LIN {X 0,Y 545.057,Z 405.592,A -85,B 0,C 180,E1 -3721.915,E2 -3721.915} C_VEL
LIN {X 0,Y 545.061,Z 405.586,A -85,B 0,C 180,E1 -3724.565,E2 -3724.565} C_VEL
LIN {X 0,Y 545.033,Z 405.597,A -85,B 0,C 180,E1 -3727.304,E2 -3727.304} C_VEL
LIN {X 0,Y 545.067,Z 405.586,A -85,B 0,C 180,E1 -3730.143,E2 -3730.143} C_VEL
LIN {X 0,Y 545.05,Z 405.588,A -85,B 0,C 180,E1 -3732.695,E2 -3732.695} C_VEL
LIN {X 0,Y 545.063,Z 405.593,A -85,B 0,C 180,E1 -3735.167,E2 -3735.167} C_VEL
LIN {X 0,Y 545.08,Z 405.583,A -85,B 0,C 180,E1 -3737.897,E2 -3737.897} C_VEL
LIN {X 0,Y 545.083,Z 405.588,A -85,B 0,C 180,E1 -3740.818,E2 -3740.818} C_VEL
LIN {X 0,Y 545.045,Z 405.589,A -85,B 0,C 180,E1 -3743.62,E2 -3743.62} C_VEL
LIN {X 0,Y 545.069,Z 405.585,A -85,B 0,C 180,E1 -3746.328,E2 -3746.328} C_VEL
LIN {X 0,Y 545.069,Z 405.593,A -85,B 0,C 180,E1 -3748.952,E2 -3748.952} C_VEL
LIN {X 0,Y 545.087,Z 405.584,A -85,B 0,C 180,E1 -3751.507,E2 -3751.507} C_VEL
LIN {X 0,Y 545.089,Z 405.589,A -85,B 0,C 180,E1 -3754.493,E2 -3754.493} C_VEL
LIN {X 0,Y 545.041,Z 405.591,A -85,B 0,C 180,E1 -3757.242,E2 -3757.242} C_VEL
LIN {X 0,Y 545.119,Z 405.586,A -85,B 0,C 180,E1 -3760.415,E2 -3760.415} C_VEL
LIN {X 0,Y 545.048,Z 405.589,A -85,B 0,C 180,E1 -3763.52,E2 -3763.52} C_VEL
LIN {X 0,Y 545.109,Z 405.613,A -85,B 0,C 180,E1 -3765.555,E2 -3765.555} C_VEL
LIN {X 0,Y 546.501,Z 411.192,A -85,B 0,C 180,E1 -3765.668,E2 -3765.668} C_VEL
LIN {X 0,Y 546.206,Z 507.654,A -85,B 0,C 180,E1 -3766.963,E2 -3766.963} C_VEL
LIN {X 0,Y 546.091,Z 520.598,A -85,B 0,C 180,E1 -3767.268,E2 -3767.268} C_VEL
LIN {X 0,Y 545.891,Z 533.301,A -85,B 0,C 180,E1 -3767.735,E2 -3767.735} C_VEL
LIN {X 0,Y 545.749,Z 543.256,A -85,B 0,C 180,E1 -3768.218,E2 -3768.218} C_VEL
LIN {X 0,Y 545.618,Z 552.755,A -85,B 0,C 180,E1 -3768.79,E2 -3768.79} C_VEL
LIN {X 0,Y 545.433,Z 561.441,A -85,B 0,C 180,E1 -3769.42,E2 -3769.42} C_VEL
LIN {X 0,Y 545.222,Z 570.054,A -85,B 0,C 180,E1 -3770.166,E2 -3770.166} C_VEL
LIN {X 0,Y 545.101,Z 577.313,A -85,B 0,C 180,E1 -3770.913,E2 -3770.913} C_VEL
LIN {X 0,Y 544.944,Z 584.959,A -85,B 0,C 180,E1 -3771.844,E2 -3771.844} C_VEL
LIN {X 0,Y 544.822,Z 592.495,A -85,B 0,C 180,E1 -3772.961,E2 -3772.961} C_VEL
LIN {X 0,Y 544.778,Z 598.448,A -85,B 0,C 180,E1 -3774.076,E2 -3774.076} C_VEL
LIN {X 0,Y 544.628,Z 603.158,A -85,B 0,C 180,E1 -3775.189,E2 -3775.189} C_VEL
LIN {X 0,Y 544.669,Z 606.782,A -85,B 0,C 180,E1 -3776.301,E2 -3776.301} C_VEL
LIN {X 0,Y 544.65,Z 608.686,A -85,B 0,C 180,E1 -3777.041,E2 -3777.041} C_VEL
LIN {X 0,Y 544.571,Z 610.122,A -85,B 0,C 180,E1 -3777.781,E2 -3777.781} C_VEL
LIN {X 0,Y 544.542,Z 611.732,A -85,B 0,C 180,E1 -3779.261,E2 -3779.261} C_VEL
LIN {X 0,Y 544.542,Z 611.996,A -85,B 0,C 180,E1 -3780,E2 -3780} C_VEL
LIN {X 0,Y 544.546,Z 611.194,A -85,B 0,C 180,E1 -3781.479,E2 -3781.479} C_VEL
LIN {X 0,Y 544.572,Z 610.282,A -85,B 0,C 180,E1 -3782.219,E2 -3782.219} C_VEL
LIN {X 0,Y 544.651,Z 608.857,A -85,B 0,C 180,E1 -3782.959,E2 -3782.959} C_VEL
LIN {X 0,Y 544.66,Z 604.819,A -85,B 0,C 180,E1 -3784.44,E2 -3784.44} C_VEL
LIN {X 0,Y 544.737,Z 600.525,A -85,B 0,C 180,E1 -3785.553,E2 -3785.553} C_VEL
LIN {X 0,Y 544.753,Z 595.248,A -85,B 0,C 180,E1 -3786.632,E2 -3786.632} C_VEL
LIN {X 0,Y 544.85,Z 589.471,A -85,B 0,C 180,E1 -3787.598,E2 -3787.598} C_VEL
LIN {X 0,Y 544.991,Z 582.775,A -85,B 0,C 180,E1 -3788.528,E2 -3788.528} C_VEL
LIN {X 0,Y 545.142,Z 574.737,A -85,B 0,C 180,E1 -3789.461,E2 -3789.461} C_VEL
LIN {X 0,Y 545.384,Z 563.744,A -85,B 0,C 180,E1 -3790.487,E2 -3790.487} C_VEL
LIN {X 0,Y 545.553,Z 554.098,A -85,B 0,C 180,E1 -3791.211,E2 -3791.211} C_VEL
LIN {X 0,Y 545.718,Z 544.947,A -85,B 0,C 180,E1 -3791.778,E2 -3791.778} C_VEL
LIN {X 0,Y 545.842,Z 535.282,A -85,B 0,C 180,E1 -3792.266,E2 -3792.266} C_VEL
LIN {X 0,Y 545.982,Z 525.933,A -85,B 0,C 180,E1 -3792.64,E2 -3792.64} C_VEL
LIN {X 0,Y 546.169,Z 515.062,A -85,B 0,C 180,E1 -3792.967,E2 -3792.967} C_VEL
LIN {X 0,Y 546.272,Z 503.356,A -85,B 0,C 180,E1 -3793.201,E2 -3793.201} C_VEL
LIN {X 0,Y 546.42,Z 410.595,A -85,B 0,C 180,E1 -3794.432,E2 -3794.432} C_VEL
LIN {X 0,Y 545.081,Z 405.586,A -85,B 0,C 180,E1 -3794.538,E2 -3794.538} C_VEL
LIN {X 0,Y 545.063,Z 405.593,A -85,B 0,C 180,E1 -3797.417,E2 -3797.417} C_VEL
LIN {X 0,Y 545.094,Z 405.583,A -85,B 0,C 180,E1 -3800.372,E2 -3800.372} C_VEL
LIN {X 0,Y 545.058,Z 405.589,A -85,B 0,C 180,E1 -3803.353,E2 -3803.353} C_VEL
LIN {X 0,Y 544.433,Z 405.67,A -85,B 0,C 180,E1 -3803.97,E2 -3803.97} C_VEL
LIN {X 0,Y 541.586,Z 406.023,A -85,B 0,C 180,E1 -3804.971,E2 -3804.971} C_VEL
LIN {X 0,Y 539.155,Z 406.323,A -85,B 0,C 180,E1 -3805.777,E2 -3805.777} C_VEL
LIN {X 0,Y 538.11,Z 406.451,A -85,B 0,C 180,E1 -3806.4,E2 -3806.4} C_VEL
LIN {X 0,Y 538.026,Z 406.462,A -85,B 0,C 180,E1 -3806.611,E2 -3806.611} C_VEL
LIN {X 0,Y 538.033,Z 406.464,A -85,B 0,C 180,E1 -3808.933,E2 -3808.933} C_VEL
LIN {X 0,Y 538.013,Z 406.461,A -85,B 0,C 180,E1 -3811.887,E2 -3811.887} C_VEL
LIN {X 0,Y 538.015,Z 406.46,A -85,B 0,C 180,E1 -3814.618,E2 -3814.618} C_VEL
LIN {X 0,Y 538.008,Z 406.471,A -85,B 0,C 180,E1 -3817.17,E2 -3817.17} C_VEL
LIN {X 0,Y 538.026,Z 406.458,A -85,B 0,C 180,E1 -3819.797,E2 -3819.797} C_VEL
LIN {X 0,Y 538.023,Z 406.47,A -85,B 0,C 180,E1 -3822.786,E2 -3822.786} C_VEL
LIN {X 0,Y 538.027,Z 406.458,A -85,B 0,C 180,E1 -3825.926,E2 -3825.926} C_VEL
LIN {X 0,Y 538.051,Z 406.458,A -85,B 0,C 180,E1 -3829.224,E2 -3829.224} C_VEL
LIN {X 0,Y 537.991,Z 406.469,A -85,B 0,C 180,E1 -3832.122,E2 -3832.122} C_VEL
LIN {X 0,Y 537.997,Z 406.469,A -85,B 0,C 180,E1 -3834.915,E2 -3834.915} C_VEL
LIN {X 0,Y 538.021,Z 406.463,A -85,B 0,C 180,E1 -3837.617,E2 -3837.617} C_VEL
LIN {X 0,Y 538.003,Z 406.473,A -85,B 0,C 180,E1 -3840.238,E2 -3840.238} C_VEL
LIN {X 0,Y 538.004,Z 406.471,A -85,B 0,C 180,E1 -3842.793,E2 -3842.793} C_VEL
LIN {X 0,Y 538.05,Z 406.63,A -85,B 0,C 180,E1 -3845.845,E2 -3845.845} C_VEL
LIN {X 0,Y 539.322,Z 413.916,A -85,B 0,C 180,E1 -3846.987,E2 -3846.987} C_VEL
LIN {X 0,Y 539.029,Z 433.076,A -85,B 0,C 180,E1 -3849.844,E2 -3849.844} C_VEL
LIN {X 0,Y 538.696,Z 451.251,A -85,B 0,C 180,E1 -3852.538,E2 -3852.538} C_VEL
LIN {X 0,Y 538.403,Z 469.786,A -85,B 0,C 180,E1 -3855.289,E2 -3855.289} C_VEL
LIN {X 0,Y 539.611,Z 479.031,A -85,B 0,C 180,E1 -3855.452,E2 -3855.452} C_VEL
LIN {X 0,Y 539.309,Z 577.904,A -85,B 0,C 180,E1 -3856.794,E2 -3856.794} C_VEL
LIN {X 0,Y 539.12,Z 590.556,A -85,B 0,C 180,E1 -3857.1,E2 -3857.1} C_VEL
LIN {X 0,Y 538.931,Z 604.503,A -85,B 0,C 180,E1 -3857.622,E2 -3857.622} C_VEL
LIN {X 0,Y 538.715,Z 615.627,A -85,B 0,C 180,E1 -3858.196,E2 -3858.196} C_VEL
LIN {X 0,Y 538.565,Z 625.158,A -85,B 0,C 180,E1 -3858.807,E2 -3858.807} C_VEL
LIN {X 0,Y 538.391,Z 633.75,A -85,B 0,C 180,E1 -3859.47,E2 -3859.47} C_VEL
LIN {X 0,Y 538.137,Z 641.979,A -85,B 0,C 180,E1 -3860.225,E2 -3860.225} C_VEL
LIN {X 0,Y 538.032,Z 648.968,A -85,B 0,C 180,E1 -3860.982,E2 -3860.982} C_VEL
LIN {X 0,Y 537.861,Z 656.298,A -85,B 0,C 180,E1 -3861.925,E2 -3861.925} C_VEL
LIN {X 0,Y 537.744,Z 662.412,A -85,B 0,C 180,E1 -3862.868,E2 -3862.868} C_VEL
LIN {X 0,Y 537.651,Z 666.834,A -85,B 0,C 180,E1 -3863.667,E2 -3863.667} C_VEL
LIN {X 0,Y 537.587,Z 671.72,A -85,B 0,C 180,E1 -3864.749,E2 -3864.749} C_VEL
LIN {X 0,Y 537.603,Z 675.698,A -85,B 0,C 180,E1 -3865.877,E2 -3865.877} C_VEL
LIN {X 0,Y 537.551,Z 678.648,A -85,B 0,C 180,E1 -3867.002,E2 -3867.002} C_VEL
LIN {X 0,Y 537.49,Z 680.143,A -85,B 0,C 180,E1 -3867.752,E2 -3867.752} C_VEL
LIN {X 0,Y 537.442,Z 681.717,A -85,B 0,C 180,E1 -3869.251,E2 -3869.251} C_VEL
LIN {X 0,Y 537.442,Z 681.996,A -85,B 0,C 180,E1 -3870,E2 -3870} C_VEL
LIN {X 0,Y 537.452,Z 681.199,A -85,B 0,C 180,E1 -3871.499,E2 -3871.499} C_VEL
LIN {X 0,Y 537.49,Z 680.28,A -85,B 0,C 180,E1 -3872.248,E2 -3872.248} C_VEL
LIN {X 0,Y 537.591,Z 677.037,A -85,B 0,C 180,E1 -3873.748,E2 -3873.748} C_VEL
LIN {X 0,Y 537.54,Z 673.478,A -85,B 0,C 180,E1 -3874.875,E2 -3874.875} C_VEL
LIN {X 0,Y 537.672,Z 670.584,A -85,B 0,C 180,E1 -3875.626,E2 -3875.626} C_VEL
LIN {X 0,Y 537.706,Z 665.105,A -85,B 0,C 180,E1 -3876.756,E2 -3876.756} C_VEL
LIN {X 0,Y 537.829,Z 658.226,A -85,B 0,C 180,E1 -3877.886,E2 -3877.886} C_VEL
LIN {X 0,Y 537.956,Z 651.262,A -85,B 0,C 180,E1 -3878.83,E2 -3878.83} C_VEL
LIN {X 0,Y 538.11,Z 644.698,A -85,B 0,C 180,E1 -3879.586,E2 -3879.586} C_VEL
LIN {X 0,Y 538.274,Z 636.977,A -85,B 0,C 180,E1 -3880.342,E2 -3880.342} C_VEL
LIN {X 0,Y 538.501,Z 627.706,A -85,B 0,C 180,E1 -3881.099,E2 -3881.099} C_VEL
LIN {X 0,Y 538.688,Z 618.38,A -85,B 0,C 180,E1 -3881.729,E2 -3881.729} C_VEL
LIN {X 0,Y 538.849,Z 609.277,A -85,B 0,C 180,E1 -3882.236,E2 -3882.236} C_VEL
LIN {X 0,Y 539.03,Z 598.562,A -85,B 0,C 180,E1 -3882.71,E2 -3882.71} C_VEL
LIN {X 0,Y 539.178,Z 586.982,A -85,B 0,C 180,E1 -3883.09,E2 -3883.09} C_VEL
LIN {X 0,Y 539.35,Z 574.949,A -85,B 0,C 180,E1 -3883.349,E2 -3883.349} C_VEL
LIN {X 0,Y 539.633,Z 477.878,A -85,B 0,C 180,E1 -3884.653,E2 -3884.653} C_VEL
LIN {X 0,Y 538.415,Z 469.73,A -85,B 0,C 180,E1 -3884.811,E2 -3884.811} C_VEL
LIN {X 0,Y 538.775,Z 447.637,A -85,B 0,C 180,E1 -3888.09,E2 -3888.09} C_VEL
LIN {X 0,Y 539.079,Z 429.341,A -85,B 0,C 180,E1 -3890.809,E2 -3890.809} C_VEL
LIN {X 0,Y 539.333,Z 414.54,A -85,B 0,C 180,E1 -3893.012,E2 -3893.012} C_VEL
LIN {X 0,Y 538.002,Z 406.471,A -85,B 0,C 180,E1 -3894.298,E2 -3894.298} C_VEL
LIN {X 0,Y 538.003,Z 406.471,A -85,B 0,C 180,E1 -3897.34,E2 -3897.34} C_VEL
LIN {X 0,Y 538.003,Z 406.473,A -85,B 0,C 180,E1 -3899.762,E2 -3899.762} C_VEL
LIN {X 0,Y 538.021,Z 406.464,A -85,B 0,C 180,E1 -3902.383,E2 -3902.383} C_VEL
LIN {X 0,Y 537.997,Z 406.471,A -85,B 0,C 180,E1 -3905.085,E2 -3905.085} C_VEL
LIN {X 0,Y 537.992,Z 406.468,A -85,B 0,C 180,E1 -3907.878,E2 -3907.878} C_VEL
LIN {X 0,Y 538.051,Z 406.46,A -85,B 0,C 180,E1 -3910.776,E2 -3910.776} C_VEL
LIN {X 0,Y 538.034,Z 406.459,A -85,B 0,C 180,E1 -3914.075,E2 -3914.075} C_VEL
LIN {X 0,Y 538.029,Z 406.468,A -85,B 0,C 180,E1 -3917.012,E2 -3917.012} C_VEL
LIN {X 0,Y 538.052,Z 406.462,A -85,B 0,C 180,E1 -3919.253,E2 -3919.253} C_VEL
LIN {X 0,Y 537.993,Z 406.467,A -85,B 0,C 180,E1 -3922.122,E2 -3922.122} C_VEL
LIN {X 0,Y 537.998,Z 406.47,A -85,B 0,C 180,E1 -3924.915,E2 -3924.915} C_VEL
LIN {X 0,Y 538.021,Z 406.462,A -85,B 0,C 180,E1 -3927.617,E2 -3927.617} C_VEL
LIN {X 0,Y 538.003,Z 406.47,A -85,B 0,C 180,E1 -3930.238,E2 -3930.238} C_VEL
LIN {X 0,Y 538.013,Z 406.468,A -85,B 0,C 180,E1 -3932.793,E2 -3932.793} C_VEL
LIN {X 0,Y 538.018,Z 406.563,A -85,B 0,C 180,E1 -3935.815,E2 -3935.815} C_VEL
LIN {X 0,Y 539.339,Z 414.074,A -85,B 0,C 180,E1 -3936.988,E2 -3936.988} C_VEL
LIN {X 0,Y 539.05,Z 431.921,A -85,B 0,C 180,E1 -3939.679,E2 -3939.679} C_VEL
LIN {X 0,Y 538.681,Z 452.563,A -85,B 0,C 180,E1 -3942.734,E2 -3942.734} C_VEL
LIN {X 0,Y 538.404,Z 469.886,A -85,B 0,C 180,E1 -3945.304,E2 -3945.304} C_VEL
LIN {X 0,Y 539.606,Z 478.79,A -85,B 0,C 180,E1 -3945.455,E2 -3945.455} C_VEL
LIN {X 0,Y 539.3,Z 576.13,A -85,B 0,C 180,E1 -3946.769,E2 -3946.769} C_VEL
LIN {X 0,Y 539.191,Z 586.049,A -85,B 0,C 180,E1 -3946.982,E2 -3946.982} C_VEL
LIN {X 0,Y 539.057,Z 596.036,A -85,B 0,C 180,E1 -3947.29,E2 -3947.29} C_VEL
LIN {X 0,Y 538.879,Z 605.384,A -85,B 0,C 180,E1 -3947.669,E2 -3947.669} C_VEL
LIN {X 0,Y 538.733,Z 615.228,A -85,B 0,C 180,E1 -3948.174,E2 -3948.174} C_VEL
LIN {X 0,Y 538.592,Z 623.796,A -85,B 0,C 180,E1 -3948.712,E2 -3948.712} C_VEL
LIN {X 0,Y 538.369,Z 632.608,A -85,B 0,C 180,E1 -3949.374,E2 -3949.374} C_VEL
LIN {X 0,Y 538.213,Z 640.052,A -85,B 0,C 180,E1 -3950.037,E2 -3950.037} C_VEL
LIN {X 0,Y 538.056,Z 647.305,A -85,B 0,C 180,E1 -3950.793,E2 -3950.793} C_VEL
LIN {X 0,Y 537.884,Z 654.929,A -85,B 0,C 180,E1 -3951.736,E2 -3951.736} C_VEL
LIN {X 0,Y 537.759,Z 661.273,A -85,B 0,C 180,E1 -3952.679,E2 -3952.679} C_VEL
LIN {X 0,Y 537.639,Z 666.854,A -85,B 0,C 180,E1 -3953.679,E2 -3953.679} C_VEL
LIN {X 0,Y 537.586,Z 671.701,A -85,B 0,C 180,E1 -3954.749,E2 -3954.749} C_VEL
LIN {X 0,Y 537.604,Z 675.701,A -85,B 0,C 180,E1 -3955.877,E2 -3955.877} C_VEL
LIN {X 0,Y 537.551,Z 678.665,A -85,B 0,C 180,E1 -3957.002,E2 -3957.002} C_VEL
LIN {X 0,Y 537.451,Z 681.145,A -85,B 0,C 180,E1 -3958.501,E2 -3958.501} C_VEL
LIN {X 0,Y 537.442,Z 681.741,A -85,B 0,C 180,E1 -3959.251,E2 -3959.251} C_VEL
LIN {X 0,Y 537.442,Z 681.806,A -85,B 0,C 180,E1 -3960.749,E2 -3960.749} C_VEL
LIN {X 0,Y 537.452,Z 681.221,A -85,B 0,C 180,E1 -3961.499,E2 -3961.499} C_VEL
LIN {X 0,Y 537.552,Z 678.878,A -85,B 0,C 180,E1 -3962.998,E2 -3962.998} C_VEL
LIN {X 0,Y 537.604,Z 675.992,A -85,B 0,C 180,E1 -3964.123,E2 -3964.123} C_VEL
LIN {X 0,Y 537.587,Z 672.073,A -85,B 0,C 180,E1 -3965.251,E2 -3965.251} C_VEL
LIN {X 0,Y 537.639,Z 667.317,A -85,B 0,C 180,E1 -3966.32,E2 -3966.32} C_VEL
LIN {X 0,Y 537.754,Z 661.829,A -85,B 0,C 180,E1 -3967.321,E2 -3967.321} C_VEL
LIN {X 0,Y 537.875,Z 655.592,A -85,B 0,C 180,E1 -3968.264,E2 -3968.264} C_VEL
LIN {X 0,Y 537.982,Z 649.743,A -85,B 0,C 180,E1 -3969.019,E2 -3969.019} C_VEL
LIN {X 0,Y 538.129,Z 642.926,A -85,B 0,C 180,E1 -3969.775,E2 -3969.775} C_VEL
LIN {X 0,Y 538.373,Z 633.697,A -85,B 0,C 180,E1 -3970.626,E2 -3970.626} C_VEL
LIN {X 0,Y 538.555,Z 625.09,A -85,B 0,C 180,E1 -3971.288,E2 -3971.288} C_VEL
LIN {X 0,Y 538.741,Z 616.029,A -85,B 0,C 180,E1 -3971.869,E2 -3971.869} C_VEL
LIN {X 0,Y 538.893,Z 606.287,A -85,B 0,C 180,E1 -3972.379,E2 -3972.379} C_VEL
LIN {X 0,Y 539.029,Z 597.178,A -85,B 0,C 180,E1 -3972.758,E2 -3972.758} C_VEL
LIN {X 0,Y 539.161,Z 587.581,A -85,B 0,C 180,E1 -3973.066,E2 -3973.066} C_VEL
LIN {X 0,Y 539.294,Z 577.096,A -85,B 0,C 180,E1 -3973.303,E2 -3973.303} C_VEL
LIN {X 0,Y 539.655,Z 478.373,A -85,B 0,C 180,E1 -3974.639,E2 -3974.639} C_VEL
LIN {X 0,Y 538.411,Z 469.814,A -85,B 0,C 180,E1 -3974.798,E2 -3974.798} C_VEL
LIN {X 0,Y 538.633,Z 454.436,A -85,B 0,C 180,E1 -3977.072,E2 -3977.072} C_VEL
LIN {X 0,Y 539.039,Z 434.478,A -85,B 0,C 180,E1 -3980.04,E2 -3980.04} C_VEL
LIN {X 0,Y 539.172,Z 413.599,A -85,B 0,C 180,E1 -3983.02,E2 -3983.02} C_VEL
LIN {X 0,Y 538.022,Z 406.471,A -85,B 0,C 180,E1 -3984.1,E2 -3984.1} C_VEL
LIN {X 0,Y 538.003,Z 406.47,A -85,B 0,C 180,E1 -3987.207,E2 -3987.207} C_VEL
LIN {X 0,Y 538.003,Z 406.473,A -85,B 0,C 180,E1 -3989.762,E2 -3989.762} C_VEL
LIN {X 0,Y 538.021,Z 406.464,A -85,B 0,C 180,E1 -3992.383,E2 -3992.383} C_VEL
LIN {X 0,Y 537.997,Z 406.471,A -85,B 0,C 180,E1 -3995.085,E2 -3995.085} C_VEL
LIN {X 0,Y 537.992,Z 406.468,A -85,B 0,C 180,E1 -3997.878,E2 -3997.878} C_VEL
LIN {X 0,Y 538.051,Z 406.463,A -85,B 0,C 180,E1 -4000.776,E2 -4000.776} C_VEL
LIN {X 0,Y 538.033,Z 406.462,A -85,B 0,C 180,E1 -4004.075,E2 -4004.075} C_VEL
LIN {X 0,Y 538.029,Z 406.468,A -85,B 0,C 180,E1 -4007.012,E2 -4007.012} C_VEL
LIN {X 0,Y 538.051,Z 406.462,A -85,B 0,C 180,E1 -4009.253,E2 -4009.253} C_VEL
LIN {X 0,Y 537.992,Z 406.468,A -85,B 0,C 180,E1 -4012.122,E2 -4012.122} C_VEL
LIN {X 0,Y 537.997,Z 406.471,A -85,B 0,C 180,E1 -4014.915,E2 -4014.915} C_VEL
LIN {X 0,Y 538.021,Z 406.463,A -85,B 0,C 180,E1 -4017.617,E2 -4017.617} C_VEL
LIN {X 0,Y 538.002,Z 406.472,A -85,B 0,C 180,E1 -4020.238,E2 -4020.238} C_VEL
LIN {X 0,Y 538.07,Z 406.661,A -85,B 0,C 180,E1 -4023.347,E2 -4023.347} C_VEL
LIN {X 0,Y 539.845,Z 415.143,A -85,B 0,C 180,E1 -4024.557,E2 -4024.557} C_VEL
LIN {X 0,Y 539.721,Z 432.182,A -85,B 0,C 180,E1 -4026.802,E2 -4026.802} C_VEL
LIN {X 0,Y 539.23,Z 454.329,A -85,B 0,C 180,E1 -4029.653,E2 -4029.653} C_VEL
LIN {X 0,Y 538.822,Z 478.604,A -85,B 0,C 180,E1 -4032.738,E2 -4032.738} C_VEL
LIN {X 0,Y 538.509,Z 498.569,A -85,B 0,C 180,E1 -4035.244,E2 -4035.244} C_VEL
LIN {X 0,Y 539.647,Z 507.696,A -85,B 0,C 180,E1 -4035.395,E2 -4035.395} C_VEL
LIN {X 0,Y 539.307,Z 607.943,A -85,B 0,C 180,E1 -4036.746,E2 -4036.746} C_VEL
LIN {X 0,Y 539.114,Z 621.214,A -85,B 0,C 180,E1 -4037.076,E2 -4037.076} C_VEL
LIN {X 0,Y 538.933,Z 633.367,A -85,B 0,C 180,E1 -4037.527,E2 -4037.527} C_VEL
LIN {X 0,Y 538.742,Z 645.405,A -85,B 0,C 180,E1 -4038.13,E2 -4038.13} C_VEL
LIN {X 0,Y 538.506,Z 657.192,A -85,B 0,C 180,E1 -4038.901,E2 -4038.901} C_VEL
LIN {X 0,Y 538.261,Z 667.604,A -85,B 0,C 180,E1 -4039.753,E2 -4039.753} C_VEL
LIN {X 0,Y 538.068,Z 676.113,A -85,B 0,C 180,E1 -4040.603,E2 -4040.603} C_VEL
LIN {X 0,Y 537.921,Z 683.96,A -85,B 0,C 180,E1 -4041.548,E2 -4041.548} C_VEL
LIN {X 0,Y 537.755,Z 691.621,A -85,B 0,C 180,E1 -4042.679,E2 -4042.679} C_VEL
LIN {X 0,Y 537.693,Z 698.679,A -85,B 0,C 180,E1 -4043.998,E2 -4043.998} C_VEL
LIN {X 0,Y 537.54,Z 703.373,A -85,B 0,C 180,E1 -4045.125,E2 -4045.125} C_VEL
LIN {X 0,Y 537.591,Z 706.958,A -85,B 0,C 180,E1 -4046.252,E2 -4046.252} C_VEL
LIN {X 0,Y 537.551,Z 708.807,A -85,B 0,C 180,E1 -4047.002,E2 -4047.002} C_VEL
LIN {X 0,Y 537.451,Z 711.182,A -85,B 0,C 180,E1 -4048.501,E2 -4048.501} C_VEL
LIN {X 0,Y 537.442,Z 712,A -85,B 0,C 180,E1 -4050,E2 -4050} C_VEL
LIN {X 0,Y 537.451,Z 711.184,A -85,B 0,C 180,E1 -4051.499,E2 -4051.499} C_VEL
LIN {X 0,Y 537.551,Z 708.81,A -85,B 0,C 180,E1 -4052.998,E2 -4052.998} C_VEL
LIN {X 0,Y 537.603,Z 705.895,A -85,B 0,C 180,E1 -4054.123,E2 -4054.123} C_VEL
LIN {X 0,Y 537.587,Z 701.948,A -85,B 0,C 180,E1 -4055.251,E2 -4055.251} C_VEL
LIN {X 0,Y 537.651,Z 697.08,A -85,B 0,C 180,E1 -4056.335,E2 -4056.335} C_VEL
LIN {X 0,Y 537.791,Z 690.466,A -85,B 0,C 180,E1 -4057.509,E2 -4057.509} C_VEL
LIN {X 0,Y 537.972,Z 682.477,A -85,B 0,C 180,E1 -4058.641,E2 -4058.641} C_VEL
LIN {X 0,Y 538.145,Z 674.332,A -85,B 0,C 180,E1 -4059.585,E2 -4059.585} C_VEL
LIN {X 0,Y 538.366,Z 664.396,A -85,B 0,C 180,E1 -4060.531,E2 -4060.531} C_VEL
LIN {X 0,Y 538.583,Z 654.591,A -85,B 0,C 180,E1 -4061.288,E2 -4061.288} C_VEL
LIN {X 0,Y 538.745,Z 643.853,A -85,B 0,C 180,E1 -4061.956,E2 -4061.956} C_VEL
LIN {X 0,Y 538.979,Z 631.099,A -85,B 0,C 180,E1 -4062.568,E2 -4062.568} C_VEL
LIN {X 0,Y 539.17,Z 618.083,A -85,B 0,C 180,E1 -4063.018,E2 -4063.018} C_VEL
LIN {X 0,Y 539.32,Z 605.098,A -85,B 0,C 180,E1 -4063.302,E2 -4063.302} C_VEL
LIN {X 0,Y 539.592,Z 506.19,A -85,B 0,C 180,E1 -4064.624,E2 -4064.624} C_VEL
LIN {X 0,Y 538.478,Z 498.265,A -85,B 0,C 180,E1 -4064.774,E2 -4064.774} C_VEL
LIN {X 0,Y 538.849,Z 473.854,A -85,B 0,C 180,E1 -4067.803,E2 -4067.803} C_VEL
LIN {X 0,Y 539.201,Z 451.45,A -85,B 0,C 180,E1 -4070.605,E2 -4070.605} C_VEL
LIN {X 0,Y 539.464,Z 427.686,A -85,B 0,C 180,E1 -4073.616,E2 -4073.616} C_VEL
LIN {X 0,Y 539.64,Z 414.953,A -85,B 0,C 180,E1 -4075.247,E2 -4075.247} C_VEL
LIN {X 0,Y 538.006,Z 406.469,A -85,B 0,C 180,E1 -4076.421,E2 -4076.421} C_VEL
LIN {X 0,Y 537.994,Z 406.469,A -85,B 0,C 180,E1 -4078.926,E2 -4078.926} C_VEL
LIN {X 0,Y 538.012,Z 406.47,A -85,B 0,C 180,E1 -4081.887,E2 -4081.887} C_VEL
LIN {X 0,Y 538.01,Z 406.465,A -85,B 0,C 180,E1 -4084.617,E2 -4084.617} C_VEL
LIN {X 0,Y 538.001,Z 406.471,A -85,B 0,C 180,E1 -4087.169,E2 -4087.169} C_VEL
LIN {X 0,Y 538.024,Z 406.466,A -85,B 0,C 180,E1 -4089.797,E2 -4089.797} C_VEL
LIN {X 0,Y 538.002,Z 406.467,A -85,B 0,C 180,E1 -4092.788,E2 -4092.788} C_VEL
LIN {X 0,Y 538.028,Z 406.469,A -85,B 0,C 180,E1 -4095.14,E2 -4095.14} C_VEL
LIN {X 0,Y 538.033,Z 406.461,A -85,B 0,C 180,E1 -4098.227,E2 -4098.227} C_VEL
LIN {X 0,Y 538.016,Z 406.47,A -85,B 0,C 180,E1 -4101.17,E2 -4101.17} C_VEL
LIN {X 0,Y 537.997,Z 406.465,A -85,B 0,C 180,E1 -4104.089,E2 -4104.089} C_VEL
LIN {X 0,Y 538.033,Z 406.466,A -85,B 0,C 180,E1 -4106.727,E2 -4106.727} C_VEL
LIN {X 0,Y 538.03,Z 406.463,A -85,B 0,C 180,E1 -4109.556,E2 -4109.556} C_VEL
LIN {X 0,Y 538.053,Z 406.467,A -85,B 0,C 180,E1 -4112.65,E2 -4112.65} C_VEL
LIN {X 0,Y 538.027,Z 406.466,A -85,B 0,C 180,E1 -4115.291,E2 -4115.291} C_VEL
LIN {X 0,Y 538.019,Z 406.466,A -85,B 0,C 180,E1 -4118.042,E2 -4118.042} C_VEL
LIN {X 0,Y 538.083,Z 406.459,A -85,B 0,C 180,E1 -4120.148,E2 -4120.148} C_VEL
LIN {X 0,Y 537.999,Z 406.468,A -85,B 0,C 180,E1 -4123.298,E2 -4123.298} C_VEL
LIN {X 0,Y 538.088,Z 406.459,A -85,B 0,C 180,E1 -4125.362,E2 -4125.362} C_VEL
LIN {X 0,Y 539.715,Z 412.557,A -85,B 0,C 180,E1 -4125.498,E2 -4125.498} C_VEL
LIN {X 0,Y 539.295,Z 508.582,A -85,B 0,C 180,E1 -4126.817,E2 -4126.817} C_VEL
LIN {X 0,Y 539.156,Z 521.366,A -85,B 0,C 180,E1 -4127.125,E2 -4127.125} C_VEL
LIN {X 0,Y 538.935,Z 534.56,A -85,B 0,C 180,E1 -4127.622,E2 -4127.622} C_VEL
LIN {X 0,Y 538.801,Z 543.956,A -85,B 0,C 180,E1 -4128.089,E2 -4128.089} C_VEL
LIN {X 0,Y 538.639,Z 554.039,A -85,B 0,C 180,E1 -4128.713,E2 -4128.713} C_VEL
LIN {X 0,Y 538.45,Z 562.824,A -85,B 0,C 180,E1 -4129.376,E2 -4129.376} C_VEL
LIN {X 0,Y 538.213,Z 570.225,A -85,B 0,C 180,E1 -4130.037,E2 -4130.037} C_VEL
LIN {X 0,Y 538.081,Z 577.418,A -85,B 0,C 180,E1 -4130.793,E2 -4130.793} C_VEL
LIN {X 0,Y 537.918,Z 583.561,A -85,B 0,C 180,E1 -4131.548,E2 -4131.548} C_VEL
LIN {X 0,Y 537.756,Z 591.312,A -85,B 0,C 180,E1 -4132.679,E2 -4132.679} C_VEL
LIN {X 0,Y 537.694,Z 598.443,A -85,B 0,C 180,E1 -4133.998,E2 -4133.998} C_VEL
LIN {X 0,Y 537.54,Z 603.153,A -85,B 0,C 180,E1 -4135.125,E2 -4135.125} C_VEL
LIN {X 0,Y 537.591,Z 606.777,A -85,B 0,C 180,E1 -4136.252,E2 -4136.252} C_VEL
LIN {X 0,Y 537.551,Z 608.682,A -85,B 0,C 180,E1 -4137.002,E2 -4137.002} C_VEL
LIN {X 0,Y 537.49,Z 610.118,A -85,B 0,C 180,E1 -4137.752,E2 -4137.752} C_VEL
LIN {X 0,Y 537.442,Z 611.725,A -85,B 0,C 180,E1 -4139.251,E2 -4139.251} C_VEL
LIN {X 0,Y 537.442,Z 611.996,A -85,B 0,C 180,E1 -4140,E2 -4140} C_VEL
LIN {X 0,Y 537.452,Z 611.187,A -85,B 0,C 180,E1 -4141.499,E2 -4141.499} C_VEL
LIN {X 0,Y 537.49,Z 610.28,A -85,B 0,C 180,E1 -4142.248,E2 -4142.248} C_VEL
LIN {X 0,Y 537.552,Z 608.85,A -85,B 0,C 180,E1 -4142.998,E2 -4142.998} C_VEL
LIN {X 0,Y 537.557,Z 604.809,A -85,B 0,C 180,E1 -4144.499,E2 -4144.499} C_VEL
LIN {X 0,Y 537.671,Z 600.515,A -85,B 0,C 180,E1 -4145.626,E2 -4145.626} C_VEL
LIN {X 0,Y 537.682,Z 595.743,A -85,B 0,C 180,E1 -4146.627,E2 -4146.627} C_VEL
LIN {X 0,Y 537.799,Z 589.459,A -85,B 0,C 180,E1 -4147.698,E2 -4147.698} C_VEL
LIN {X 0,Y 537.951,Z 582.797,A -85,B 0,C 180,E1 -4148.641,E2 -4148.641} C_VEL
LIN {X 0,Y 538.131,Z 574.833,A -85,B 0,C 180,E1 -4149.585,E2 -4149.585} C_VEL
LIN {X 0,Y 538.387,Z 563.89,A -85,B 0,C 180,E1 -4150.625,E2 -4150.625} C_VEL
LIN {X 0,Y 538.563,Z 555.302,A -85,B 0,C 180,E1 -4151.288,E2 -4151.288} C_VEL
LIN {X 0,Y 538.764,Z 544.938,A -85,B 0,C 180,E1 -4151.943,E2 -4151.943} C_VEL
LIN {X 0,Y 538.911,Z 534.391,A -85,B 0,C 180,E1 -4152.474,E2 -4152.474} C_VEL
LIN {X 0,Y 539.183,Z 521.951,A -85,B 0,C 180,E1 -4152.946,E2 -4152.946} C_VEL
LIN {X 0,Y 539.274,Z 509.732,A -85,B 0,C 180,E1 -4153.255,E2 -4153.255} C_VEL
LIN {X 0,Y 539.454,Z 479.835,A -85,B 0,C 180,E1 -4153.682,E2 -4153.682} C_VEL
LIN {X 0,Y 539.592,Z 411.558,A -85,B 0,C 180,E1 -4154.605,E2 -4154.605} C_VEL
LIN {X 0,Y 538.059,Z 406.461,A -85,B 0,C 180,E1 -4154.736,E2 -4154.736} C_VEL
LIN {X 0,Y 538.015,Z 406.472,A -85,B 0,C 180,E1 -4157.524,E2 -4157.524} C_VEL
LIN {X 0,Y 538.088,Z 406.459,A -85,B 0,C 180,E1 -4159.881,E2 -4159.881} C_VEL
LIN {X 0,Y 538.014,Z 406.467,A -85,B 0,C 180,E1 -4163.072,E2 -4163.072} C_VEL
LIN {X 0,Y 538.033,Z 406.46,A -85,B 0,C 180,E1 -4166.367,E2 -4166.367} C_VEL
LIN {X 0,Y 538.026,Z 406.462,A -85,B 0,C 180,E1 -4166.611,E2 -4166.611} C_VEL
LIN {X 0,Y 537.359,Z 406.552,A -85,B 0,C 180,E1 -4167.235,E2 -4167.235} C_VEL
LIN {X 0,Y 534.492,Z 406.908,A -85,B 0,C 180,E1 -4168.249,E2 -4168.249} C_VEL
LIN {X 0,Y 532.073,Z 407.208,A -85,B 0,C 180,E1 -4169.066,E2 -4169.066} C_VEL
LIN {X 0,Y 531.042,Z 407.335,A -85,B 0,C 180,E1 -4169.696,E2 -4169.696} C_VEL
LIN {X 0,Y 530.962,Z 407.342,A -85,B 0,C 180,E1 -4169.91,E2 -4169.91} C_VEL
LIN {X 0,Y 530.97,Z 407.343,A -85,B 0,C 180,E1 -4172.867,E2 -4172.867} C_VEL
LIN {X 0,Y 530.957,Z 407.344,A -85,B 0,C 180,E1 -4175.62,E2 -4175.62} C_VEL
LIN {X 0,Y 530.97,Z 407.345,A -85,B 0,C 180,E1 -4178.654,E2 -4178.654} C_VEL
LIN {X 0,Y 530.997,Z 407.339,A -85,B 0,C 180,E1 -4181.436,E2 -4181.436} C_VEL
LIN {X 0,Y 530.989,Z 407.344,A -85,B 0,C 180,E1 -4184.547,E2 -4184.547} C_VEL
LIN {X 0,Y 530.985,Z 407.339,A -85,B 0,C 180,E1 -4187.834,E2 -4187.834} C_VEL
LIN {X 0,Y 530.988,Z 407.343,A -85,B 0,C 180,E1 -4190.556,E2 -4190.556} C_VEL
LIN {X 0,Y 530.953,Z 407.342,A -85,B 0,C 180,E1 -4193.441,E2 -4193.441} C_VEL
LIN {X 0,Y 531.002,Z 407.344,A -85,B 0,C 180,E1 -4196.494,E2 -4196.494} C_VEL
LIN {X 0,Y 530.964,Z 407.343,A -85,B 0,C 180,E1 -4199.357,E2 -4199.357} C_VEL
LIN {X 0,Y 530.963,Z 407.351,A -85,B 0,C 180,E1 -4202.479,E2 -4202.479} C_VEL
LIN {X 0,Y 531.015,Z 407.464,A -85,B 0,C 180,E1 -4205.673,E2 -4205.673} C_VEL
LIN {X 0,Y 532.36,Z 415.042,A -85,B 0,C 180,E1 -4206.874,E2 -4206.874} C_VEL
LIN {X 0,Y 532.068,Z 433.71,A -85,B 0,C 180,E1 -4209.69,E2 -4209.69} C_VEL
LIN {X 0,Y 531.696,Z 453.83,A -85,B 0,C 180,E1 -4212.698,E2 -4212.698} C_VEL
LIN {X 0,Y 531.409,Z 469.902,A -85,B 0,C 180,E1 -4215.092,E2 -4215.092} C_VEL
LIN {X 0,Y 532.745,Z 479.269,A -85,B 0,C 180,E1 -4215.262,E2 -4215.262} C_VEL
LIN {X 0,Y 532.414,Z 578.141,A -85,B 0,C 180,E1 -4216.619,E2 -4216.619} C_VEL
LIN {X 0,Y 532.207,Z 591.571,A -85,B 0,C 180,E1 -4216.954,E2 -4216.954} C_VEL
LIN {X 0,Y 532,Z 604.658,A -85,B 0,C 180,E1 -4217.458,E2 -4217.458} C_VEL
LIN {X 0,Y 531.79,Z 616.926,A -85,B 0,C 180,E1 -4218.099,E2 -4218.099} C_VEL
LIN {X 0,Y 531.549,Z 628.024,A -85,B 0,C 180,E1 -4218.851,E2 -4218.851} C_VEL
LIN {X 0,Y 531.227,Z 639.261,A -85,B 0,C 180,E1 -4219.808,E2 -4219.808} C_VEL
LIN {X 0,Y 531.023,Z 647.488,A -85,B 0,C 180,E1 -4220.67,E2 -4220.67} C_VEL
LIN {X 0,Y 530.851,Z 655.076,A -85,B 0,C 180,E1 -4221.626,E2 -4221.626} C_VEL
LIN {X 0,Y 530.672,Z 662.446,A -85,B 0,C 180,E1 -4222.772,E2 -4222.772} C_VEL
LIN {X 0,Y 530.564,Z 667.294,A -85,B 0,C 180,E1 -4223.681,E2 -4223.681} C_VEL
LIN {X 0,Y 530.524,Z 671.716,A -85,B 0,C 180,E1 -4224.679,E2 -4224.679} C_VEL
LIN {X 0,Y 530.523,Z 675.693,A -85,B 0,C 180,E1 -4225.822,E2 -4225.822} C_VEL
LIN {X 0,Y 530.457,Z 678.641,A -85,B 0,C 180,E1 -4226.962,E2 -4226.962} C_VEL
LIN {X 0,Y 530.411,Z 680.144,A -85,B 0,C 180,E1 -4227.722,E2 -4227.722} C_VEL
LIN {X 0,Y 530.344,Z 681.709,A -85,B 0,C 180,E1 -4229.241,E2 -4229.241} C_VEL
LIN {X 0,Y 530.343,Z 681.997,A -85,B 0,C 180,E1 -4230,E2 -4230} C_VEL
LIN {X 0,Y 530.361,Z 681.191,A -85,B 0,C 180,E1 -4231.519,E2 -4231.519} C_VEL
LIN {X 0,Y 530.411,Z 680.281,A -85,B 0,C 180,E1 -4232.278,E2 -4232.278} C_VEL
LIN {X 0,Y 530.516,Z 677.029,A -85,B 0,C 180,E1 -4233.798,E2 -4233.798} C_VEL
LIN {X 0,Y 530.458,Z 673.469,A -85,B 0,C 180,E1 -4234.94,E2 -4234.94} C_VEL
LIN {X 0,Y 530.605,Z 670.581,A -85,B 0,C 180,E1 -4235.701,E2 -4235.701} C_VEL
LIN {X 0,Y 530.637,Z 665.106,A -85,B 0,C 180,E1 -4236.846,E2 -4236.846} C_VEL
LIN {X 0,Y 530.778,Z 658.289,A -85,B 0,C 180,E1 -4237.992,E2 -4237.992} C_VEL
LIN {X 0,Y 530.913,Z 651.396,A -85,B 0,C 180,E1 -4238.948,E2 -4238.948} C_VEL
LIN {X 0,Y 531.11,Z 643.041,A -85,B 0,C 180,E1 -4239.906,E2 -4239.906} C_VEL
LIN {X 0,Y 531.409,Z 632.761,A -85,B 0,C 180,E1 -4240.863,E2 -4240.863} C_VEL
LIN {X 0,Y 531.673,Z 622.145,A -85,B 0,C 180,E1 -4241.661,E2 -4241.661} C_VEL
LIN {X 0,Y 531.916,Z 609.524,A -85,B 0,C 180,E1 -4242.398,E2 -4242.398} C_VEL
LIN {X 0,Y 532.151,Z 597.599,A -85,B 0,C 180,E1 -4242.926,E2 -4242.926} C_VEL
LIN {X 0,Y 532.331,Z 584.422,A -85,B 0,C 180,E1 -4243.334,E2 -4243.334} C_VEL
LIN {X 0,Y 532.476,Z 570.119,A -85,B 0,C 180,E1 -4243.598,E2 -4243.598} C_VEL
LIN {X 0,Y 532.758,Z 478.179,A -85,B 0,C 180,E1 -4244.843,E2 -4244.843} C_VEL
LIN {X 0,Y 531.426,Z 469.82,A -85,B 0,C 180,E1 -4245.009,E2 -4245.009} C_VEL
LIN {X 0,Y 531.774,Z 448.93,A -85,B 0,C 180,E1 -4248.128,E2 -4248.128} C_VEL
LIN {X 0,Y 532.112,Z 430.466,A -85,B 0,C 180,E1 -4250.892,E2 -4250.892} C_VEL
LIN {X 0,Y 532.383,Z 415.639,A -85,B 0,C 180,E1 -4253.125,E2 -4253.125} C_VEL
LIN {X 0,Y 530.96,Z 407.348,A -85,B 0,C 180,E1 -4254.46,E2 -4254.46} C_VEL
LIN {X 0,Y 530.963,Z 407.35,A -85,B 0,C 180,E1 -4257.521,E2 -4257.521} C_VEL
LIN {X 0,Y 530.964,Z 407.343,A -85,B 0,C 180,E1 -4260.643,E2 -4260.643} C_VEL
LIN {X 0,Y 530.99,Z 407.344,A -85,B 0,C 180,E1 -4263.773,E2 -4263.773} C_VEL
LIN {X 0,Y 530.953,Z 407.344,A -85,B 0,C 180,E1 -4266.559,E2 -4266.559} C_VEL
LIN {X 0,Y 530.988,Z 407.343,A -85,B 0,C 180,E1 -4269.443,E2 -4269.443} C_VEL
LIN {X 0,Y 530.981,Z 407.341,A -85,B 0,C 180,E1 -4272.457,E2 -4272.457} C_VEL
LIN {X 0,Y 530.992,Z 407.341,A -85,B 0,C 180,E1 -4275.621,E2 -4275.621} C_VEL
LIN {X 0,Y 530.997,Z 407.339,A -85,B 0,C 180,E1 -4278.564,E2 -4278.564} C_VEL
LIN {X 0,Y 530.96,Z 407.342,A -85,B 0,C 180,E1 -4281.529,E2 -4281.529} C_VEL
LIN {X 0,Y 530.953,Z 407.342,A -85,B 0,C 180,E1 -4284.38,E2 -4284.38} C_VEL
LIN {X 0,Y 530.97,Z 407.343,A -85,B 0,C 180,E1 -4287.133,E2 -4287.133} C_VEL
LIN {X 0,Y 530.954,Z 407.344,A -85,B 0,C 180,E1 -4289.802,E2 -4289.802} C_VEL
LIN {X 0,Y 530.967,Z 407.349,A -85,B 0,C 180,E1 -4292.478,E2 -4292.478} C_VEL
LIN {X 0,Y 530.986,Z 407.351,A -85,B 0,C 180,E1 -4295.646,E2 -4295.646} C_VEL
LIN {X 0,Y 532.365,Z 415.113,A -85,B 0,C 180,E1 -4296.875,E2 -4296.875} C_VEL
LIN {X 0,Y 532.097,Z 432.497,A -85,B 0,C 180,E1 -4299.498,E2 -4299.498} C_VEL
LIN {X 0,Y 531.717,Z 452.564,A -85,B 0,C 180,E1 -4302.5,E2 -4302.5} C_VEL
LIN {X 0,Y 531.395,Z 469.912,A -85,B 0,C 180,E1 -4305.103,E2 -4305.103} C_VEL
LIN {X 0,Y 532.715,Z 479.434,A -85,B 0,C 180,E1 -4305.281,E2 -4305.281} C_VEL
LIN {X 0,Y 532.382,Z 576.672,A -85,B 0,C 180,E1 -4306.619,E2 -4306.619} C_VEL
LIN {X 0,Y 532.229,Z 587.327,A -85,B 0,C 180,E1 -4306.858,E2 -4306.858} C_VEL
LIN {X 0,Y 532.075,Z 598.321,A -85,B 0,C 180,E1 -4307.218,E2 -4307.218} C_VEL
LIN {X 0,Y 531.849,Z 611.178,A -85,B 0,C 180,E1 -4307.794,E2 -4307.794} C_VEL
LIN {X 0,Y 531.661,Z 622.125,A -85,B 0,C 180,E1 -4308.45,E2 -4308.45} C_VEL
LIN {X 0,Y 531.418,Z 631.429,A -85,B 0,C 180,E1 -4309.137,E2 -4309.137} C_VEL
LIN {X 0,Y 531.204,Z 640.052,A -85,B 0,C 180,E1 -4309.904,E2 -4309.904} C_VEL
LIN {X 0,Y 531.025,Z 647.317,A -85,B 0,C 180,E1 -4310.67,E2 -4310.67} C_VEL
LIN {X 0,Y 530.849,Z 654.941,A -85,B 0,C 180,E1 -4311.626,E2 -4311.626} C_VEL
LIN {X 0,Y 530.69,Z 661.276,A -85,B 0,C 180,E1 -4312.581,E2 -4312.581} C_VEL
LIN {X 0,Y 530.598,Z 665.958,A -85,B 0,C 180,E1 -4313.42,E2 -4313.42} C_VEL
LIN {X 0,Y 530.608,Z 670.125,A -85,B 0,C 180,E1 -4314.299,E2 -4314.299} C_VEL
LIN {X 0,Y 530.462,Z 674.469,A -85,B 0,C 180,E1 -4315.441,E2 -4315.441} C_VEL
LIN {X 0,Y 530.516,Z 676.847,A -85,B 0,C 180,E1 -4316.202,E2 -4316.202} C_VEL
LIN {X 0,Y 530.457,Z 678.66,A -85,B 0,C 180,E1 -4316.962,E2 -4316.962} C_VEL
LIN {X 0,Y 530.361,Z 681.138,A -85,B 0,C 180,E1 -4318.481,E2 -4318.481} C_VEL
LIN {X 0,Y 530.344,Z 681.734,A -85,B 0,C 180,E1 -4319.241,E2 -4319.241} C_VEL
LIN {X 0,Y 530.344,Z 681.8,A -85,B 0,C 180,E1 -4320.759,E2 -4320.759} C_VEL
LIN {X 0,Y 530.361,Z 681.213,A -85,B 0,C 180,E1 -4321.519,E2 -4321.519} C_VEL
LIN {X 0,Y 530.457,Z 678.87,A -85,B 0,C 180,E1 -4323.038,E2 -4323.038} C_VEL
LIN {X 0,Y 530.523,Z 675.984,A -85,B 0,C 180,E1 -4324.178,E2 -4324.178} C_VEL
LIN {X 0,Y 530.524,Z 672.063,A -85,B 0,C 180,E1 -4325.321,E2 -4325.321} C_VEL
LIN {X 0,Y 530.553,Z 667.804,A -85,B 0,C 180,E1 -4326.306,E2 -4326.306} C_VEL
LIN {X 0,Y 530.679,Z 661.826,A -85,B 0,C 180,E1 -4327.419,E2 -4327.419} C_VEL
LIN {X 0,Y 530.839,Z 655.597,A -85,B 0,C 180,E1 -4328.374,E2 -4328.374} C_VEL
LIN {X 0,Y 530.937,Z 649.745,A -85,B 0,C 180,E1 -4329.14,E2 -4329.14} C_VEL
LIN {X 0,Y 531.103,Z 642.913,A -85,B 0,C 180,E1 -4329.906,E2 -4329.906} C_VEL
LIN {X 0,Y 531.353,Z 633.651,A -85,B 0,C 180,E1 -4330.768,E2 -4330.768} C_VEL
LIN {X 0,Y 531.584,Z 624.99,A -85,B 0,C 180,E1 -4331.438,E2 -4331.438} C_VEL
LIN {X 0,Y 531.758,Z 615.745,A -85,B 0,C 180,E1 -4332.033,E2 -4332.033} C_VEL
LIN {X 0,Y 531.902,Z 605.977,A -85,B 0,C 180,E1 -4332.544,E2 -4332.544} C_VEL
LIN {X 0,Y 532.138,Z 594.109,A -85,B 0,C 180,E1 -4333.023,E2 -4333.023} C_VEL
LIN {X 0,Y 532.341,Z 579.983,A -85,B 0,C 180,E1 -4333.407,E2 -4333.407} C_VEL
LIN {X 0,Y 532.505,Z 553.762,A -85,B 0,C 180,E1 -4333.791,E2 -4333.791} C_VEL
LIN {X 0,Y 532.715,Z 478.151,A -85,B 0,C 180,E1 -4334.826,E2 -4334.826} C_VEL
LIN {X 0,Y 531.432,Z 469.958,A -85,B 0,C 180,E1 -4334.989,E2 -4334.989} C_VEL
LIN {X 0,Y 531.673,Z 454.42,A -85,B 0,C 180,E1 -4337.303,E2 -4337.303} C_VEL
LIN {X 0,Y 531.927,Z 439.805,A -85,B 0,C 180,E1 -4339.488,E2 -4339.488} C_VEL
LIN {X 0,Y 532.203,Z 419.387,A -85,B 0,C 180,E1 -4342.424,E2 -4342.424} C_VEL
LIN {X 0,Y 532.027,Z 412.997,A -85,B 0,C 180,E1 -4343.347,E2 -4343.347} C_VEL
LIN {X 0,Y 530.981,Z 407.347,A -85,B 0,C 180,E1 -4344.193,E2 -4344.193} C_VEL
LIN {X 0,Y 530.95,Z 407.346,A -85,B 0,C 180,E1 -4346.747,E2 -4346.747} C_VEL
LIN {X 0,Y 530.964,Z 407.349,A -85,B 0,C 180,E1 -4349.324,E2 -4349.324} C_VEL
LIN {X 0,Y 530.968,Z 407.344,A -85,B 0,C 180,E1 -4352.1,E2 -4352.1} C_VEL
LIN {X 0,Y 530.97,Z 407.344,A -85,B 0,C 180,E1 -4354.851,E2 -4354.851} C_VEL
LIN {X 0,Y 530.966,Z 407.347,A -85,B 0,C 180,E1 -4357.508,E2 -4357.508} C_VEL
LIN {X 0,Y 530.983,Z 407.34,A -85,B 0,C 180,E1 -4360.433,E2 -4360.433} C_VEL
LIN {X 0,Y 530.968,Z 407.345,A -85,B 0,C 180,E1 -4363.494,E2 -4363.494} C_VEL
LIN {X 0,Y 530.968,Z 407.345,A -85,B 0,C 180,E1 -4366.505,E2 -4366.505} C_VEL
LIN {X 0,Y 530.983,Z 407.34,A -85,B 0,C 180,E1 -4369.567,E2 -4369.567} C_VEL
LIN {X 0,Y 530.968,Z 407.348,A -85,B 0,C 180,E1 -4372.577,E2 -4372.577} C_VEL
LIN {X 0,Y 530.983,Z 407.341,A -85,B 0,C 180,E1 -4375.309,E2 -4375.309} C_VEL
LIN {X 0,Y 530.969,Z 407.344,A -85,B 0,C 180,E1 -4378.032,E2 -4378.032} C_VEL
LIN {X 0,Y 530.965,Z 407.347,A -85,B 0,C 180,E1 -4380.879,E2 -4380.879} C_VEL
LIN {X 0,Y 531.005,Z 407.51,A -85,B 0,C 180,E1 -4383.15,E2 -4383.15} C_VEL
LIN {X 0,Y 533.042,Z 417.763,A -85,B 0,C 180,E1 -4384.627,E2 -4384.627} C_VEL
LIN {X 0,Y 532.613,Z 438.036,A -85,B 0,C 180,E1 -4387.317,E2 -4387.317} C_VEL
LIN {X 0,Y 532.229,Z 458.007,A -85,B 0,C 180,E1 -4389.92,E2 -4389.92} C_VEL
LIN {X 0,Y 531.764,Z 481.161,A -85,B 0,C 180,E1 -4392.898,E2 -4392.898} C_VEL
LIN {X 0,Y 531.481,Z 498.32,A -85,B 0,C 180,E1 -4395.059,E2 -4395.059} C_VEL
LIN {X 0,Y 532.748,Z 508.961,A -85,B 0,C 180,E1 -4395.237,E2 -4395.237} C_VEL
LIN {X 0,Y 532.376,Z 606.596,A -85,B 0,C 180,E1 -4396.57,E2 -4396.57} C_VEL
LIN {X 0,Y 532.196,Z 619.512,A -85,B 0,C 180,E1 -4396.881,E2 -4396.881} C_VEL
LIN {X 0,Y 531.949,Z 632.662,A -85,B 0,C 180,E1 -4397.36,E2 -4397.36} C_VEL
LIN {X 0,Y 531.744,Z 644.95,A -85,B 0,C 180,E1 -4397.974,E2 -4397.974} C_VEL
LIN {X 0,Y 531.525,Z 656.901,A -85,B 0,C 180,E1 -4398.754,E2 -4398.754} C_VEL
LIN {X 0,Y 531.233,Z 667.473,A -85,B 0,C 180,E1 -4399.615,E2 -4399.615} C_VEL
LIN {X 0,Y 531.062,Z 676.093,A -85,B 0,C 180,E1 -4400.478,E2 -4400.478} C_VEL
LIN {X 0,Y 530.887,Z 683.96,A -85,B 0,C 180,E1 -4401.435,E2 -4401.435} C_VEL
LIN {X 0,Y 530.685,Z 691.621,A -85,B 0,C 180,E1 -4402.581,E2 -4402.581} C_VEL
LIN {X 0,Y 530.604,Z 698.679,A -85,B 0,C 180,E1 -4403.917,E2 -4403.917} C_VEL
LIN {X 0,Y 530.459,Z 703.373,A -85,B 0,C 180,E1 -4405.06,E2 -4405.06} C_VEL
LIN {X 0,Y 530.516,Z 706.958,A -85,B 0,C 180,E1 -4406.202,E2 -4406.202} C_VEL
LIN {X 0,Y 530.457,Z 708.807,A -85,B 0,C 180,E1 -4406.962,E2 -4406.962} C_VEL
LIN {X 0,Y 530.411,Z 710.193,A -85,B 0,C 180,E1 -4407.722,E2 -4407.722} C_VEL
LIN {X 0,Y 530.344,Z 711.785,A -85,B 0,C 180,E1 -4409.241,E2 -4409.241} C_VEL
LIN {X 0,Y 530.342,Z 712,A -85,B 0,C 180,E1 -4410,E2 -4410} C_VEL
LIN {X 0,Y 530.361,Z 711.183,A -85,B 0,C 180,E1 -4411.519,E2 -4411.519} C_VEL
LIN {X 0,Y 530.411,Z 710.196,A -85,B 0,C 180,E1 -4412.278,E2 -4412.278} C_VEL
LIN {X 0,Y 530.457,Z 708.81,A -85,B 0,C 180,E1 -4413.038,E2 -4413.038} C_VEL
LIN {X 0,Y 530.523,Z 705.895,A -85,B 0,C 180,E1 -4414.178,E2 -4414.178} C_VEL
LIN {X 0,Y 530.524,Z 701.948,A -85,B 0,C 180,E1 -4415.321,E2 -4415.321} C_VEL
LIN {X 0,Y 530.599,Z 696.262,A -85,B 0,C 180,E1 -4416.582,E2 -4416.582} C_VEL
LIN {X 0,Y 530.758,Z 689.235,A -85,B 0,C 180,E1 -4417.801,E2 -4417.801} C_VEL
LIN {X 0,Y 530.93,Z 680.991,A -85,B 0,C 180,E1 -4418.948,E2 -4418.948} C_VEL
LIN {X 0,Y 531.139,Z 672.485,A -85,B 0,C 180,E1 -4419.905,E2 -4419.905} C_VEL
LIN {X 0,Y 531.377,Z 661.852,A -85,B 0,C 180,E1 -4420.864,E2 -4420.864} C_VEL
LIN {X 0,Y 531.661,Z 650.926,A -85,B 0,C 180,E1 -4421.656,E2 -4421.656} C_VEL
LIN {X 0,Y 531.862,Z 639.71,A -85,B 0,C 180,E1 -4422.303,E2 -4422.303} C_VEL
LIN {X 0,Y 532.057,Z 627.754,A -85,B 0,C 180,E1 -4422.831,E2 -4422.831} C_VEL
LIN {X 0,Y 532.279,Z 613.961,A -85,B 0,C 180,E1 -4423.263,E2 -4423.263} C_VEL
LIN {X 0,Y 532.421,Z 601.608,A -85,B 0,C 180,E1 -4423.502,E2 -4423.502} C_VEL
LIN {X 0,Y 532.698,Z 507.195,A -85,B 0,C 180,E1 -4424.779,E2 -4424.779} C_VEL
LIN {X 0,Y 531.435,Z 497.415,A -85,B 0,C 180,E1 -4424.972,E2 -4424.972} C_VEL
LIN {X 0,Y 531.824,Z 473.953,A -85,B 0,C 180,E1 -4427.922,E2 -4427.922} C_VEL
LIN {X 0,Y 532.247,Z 448.992,A -85,B 0,C 180,E1 -4431.089,E2 -4431.089} C_VEL
LIN {X 0,Y 532.633,Z 423.794,A -85,B 0,C 180,E1 -4434.333,E2 -4434.333} C_VEL
LIN {X 0,Y 532.624,Z 415.704,A -85,B 0,C 180,E1 -4435.394,E2 -4435.394} C_VEL
LIN {X 0,Y 530.958,Z 407.347,A -85,B 0,C 180,E1 -4436.594,E2 -4436.594} C_VEL
LIN {X 0,Y 530.963,Z 407.349,A -85,B 0,C 180,E1 -4439.324,E2 -4439.324} C_VEL
LIN {X 0,Y 530.967,Z 407.345,A -85,B 0,C 180,E1 -4442.1,E2 -4442.1} C_VEL
LIN {X 0,Y 530.968,Z 407.343,A -85,B 0,C 180,E1 -4444.85,E2 -4444.85} C_VEL
LIN {X 0,Y 530.965,Z 407.349,A -85,B 0,C 180,E1 -4447.508,E2 -4447.508} C_VEL
LIN {X 0,Y 530.983,Z 407.34,A -85,B 0,C 180,E1 -4450.433,E2 -4450.433} C_VEL
LIN {X 0,Y 530.947,Z 407.35,A -85,B 0,C 180,E1 -4453.497,E2 -4453.497} C_VEL
LIN {X 0,Y 530.958,Z 407.344,A -85,B 0,C 180,E1 -4456.504,E2 -4456.504} C_VEL
LIN {X 0,Y 530.987,Z 407.345,A -85,B 0,C 180,E1 -4458.976,E2 -4458.976} C_VEL
LIN {X 0,Y 530.96,Z 407.345,A -85,B 0,C 180,E1 -4461.529,E2 -4461.529} C_VEL
LIN {X 0,Y 530.958,Z 407.344,A -85,B 0,C 180,E1 -4464.38,E2 -4464.38} C_VEL
LIN {X 0,Y 530.97,Z 407.347,A -85,B 0,C 180,E1 -4467.133,E2 -4467.133} C_VEL
LIN {X 0,Y 530.972,Z 407.341,A -85,B 0,C 180,E1 -4469.803,E2 -4469.803} C_VEL
LIN {X 0,Y 531.014,Z 407.341,A -85,B 0,C 180,E1 -4472.468,E2 -4472.468} C_VEL
LIN {X 0,Y 530.992,Z 407.346,A -85,B 0,C 180,E1 -4474.942,E2 -4474.942} C_VEL
LIN {X 0,Y 530.975,Z 407.346,A -85,B 0,C 180,E1 -4478.247,E2 -4478.247} C_VEL
LIN {X 0,Y 530.986,Z 407.347,A -85,B 0,C 180,E1 -4480.677,E2 -4480.677} C_VEL
LIN {X 0,Y 530.962,Z 407.347,A -85,B 0,C 180,E1 -4483.07,E2 -4483.07} C_VEL
LIN {X 0,Y 531.025,Z 407.34,A -85,B 0,C 180,E1 -4485.173,E2 -4485.173} C_VEL
LIN {X 0,Y 532.79,Z 412.89,A -85,B 0,C 180,E1 -4485.306,E2 -4485.306} C_VEL
LIN {X 0,Y 532.386,Z 509.48,A -85,B 0,C 180,E1 -4486.667,E2 -4486.667} C_VEL
LIN {X 0,Y 532.199,Z 522.854,A -85,B 0,C 180,E1 -4487.003,E2 -4487.003} C_VEL
LIN {X 0,Y 532.01,Z 534.846,A -85,B 0,C 180,E1 -4487.459,E2 -4487.459} C_VEL
LIN {X 0,Y 531.829,Z 545.693,A -85,B 0,C 180,E1 -4488.009,E2 -4488.009} C_VEL
LIN {X 0,Y 531.65,Z 555.867,A -85,B 0,C 180,E1 -4488.66,E2 -4488.66} C_VEL
LIN {X 0,Y 531.358,Z 566.735,A -85,B 0,C 180,E1 -4489.522,E2 -4489.522} C_VEL
LIN {X 0,Y 531.129,Z 576.325,A -85,B 0,C 180,E1 -4490.479,E2 -4490.479} C_VEL
LIN {X 0,Y 530.919,Z 584.168,A -85,B 0,C 180,E1 -4491.436,E2 -4491.436} C_VEL
LIN {X 0,Y 530.781,Z 590.68,A -85,B 0,C 180,E1 -4492.391,E2 -4492.391} C_VEL
LIN {X 0,Y 530.664,Z 596.159,A -85,B 0,C 180,E1 -4493.358,E2 -4493.358} C_VEL
LIN {X 0,Y 530.614,Z 600.566,A -85,B 0,C 180,E1 -4494.299,E2 -4494.299} C_VEL
LIN {X 0,Y 530.505,Z 604.874,A -85,B 0,C 180,E1 -4495.441,E2 -4495.441} C_VEL
LIN {X 0,Y 530.516,Z 607.12,A -85,B 0,C 180,E1 -4496.202,E2 -4496.202} C_VEL
LIN {X 0,Y 530.486,Z 608.99,A -85,B 0,C 180,E1 -4496.962,E2 -4496.962} C_VEL
LIN {X 0,Y 530.411,Z 610.401,A -85,B 0,C 180,E1 -4497.722,E2 -4497.722} C_VEL
LIN {X 0,Y 530.347,Z 611.978,A -85,B 0,C 180,E1 -4499.241,E2 -4499.241} C_VEL
LIN {X 0,Y 530.347,Z 612.24,A -85,B 0,C 180,E1 -4500,E2 -4500} C_VEL
LIN {X 0,Y 530.361,Z 611.437,A -85,B 0,C 180,E1 -4501.519,E2 -4501.519} C_VEL
LIN {X 0,Y 530.411,Z 610.538,A -85,B 0,C 180,E1 -4502.278,E2 -4502.278} C_VEL
LIN {X 0,Y 530.487,Z 609.132,A -85,B 0,C 180,E1 -4503.038,E2 -4503.038} C_VEL
LIN {X 0,Y 530.485,Z 605.145,A -85,B 0,C 180,E1 -4504.559,E2 -4504.559} C_VEL
LIN {X 0,Y 530.606,Z 600.9,A -85,B 0,C 180,E1 -4505.701,E2 -4505.701} C_VEL
LIN {X 0,Y 530.639,Z 596.627,A -85,B 0,C 180,E1 -4506.63,E2 -4506.63} C_VEL
LIN {X 0,Y 530.755,Z 591.161,A -85,B 0,C 180,E1 -4507.609,E2 -4507.609} C_VEL
LIN {X 0,Y 530.905,Z 584.732,A -85,B 0,C 180,E1 -4508.565,E2 -4508.565} C_VEL
LIN {X 0,Y 531.076,Z 576.989,A -85,B 0,C 180,E1 -4509.522,E2 -4509.522} C_VEL
LIN {X 0,Y 531.332,Z 567.6,A -85,B 0,C 180,E1 -4510.479,E2 -4510.479} C_VEL
LIN {X 0,Y 531.589,Z 557.033,A -85,B 0,C 180,E1 -4511.342,E2 -4511.342} C_VEL
LIN {X 0,Y 531.832,Z 545.743,A -85,B 0,C 180,E1 -4512.07,E2 -4512.07} C_VEL
LIN {X 0,Y 531.989,Z 534.592,A -85,B 0,C 180,E1 -4512.639,E2 -4512.639} C_VEL
LIN {X 0,Y 532.284,Z 521.137,A -85,B 0,C 180,E1 -4513.141,E2 -4513.141} C_VEL
LIN {X 0,Y 532.371,Z 507.983,A -85,B 0,C 180,E1 -4513.455,E2 -4513.455} C_VEL
LIN {X 0,Y 532.746,Z 412.885,A -85,B 0,C 180,E1 -4514.779,E2 -4514.779} C_VEL
LIN {X 0,Y 531.01,Z 407.341,A -85,B 0,C 180,E1 -4514.915,E2 -4514.915} C_VEL
LIN {X 0,Y 530.975,Z 407.349,A -85,B 0,C 180,E1 -4517.724,E2 -4517.724} C_VEL
LIN {X 0,Y 531.028,Z 407.336,A -85,B 0,C 180,E1 -4520.127,E2 -4520.127} C_VEL
LIN {X 0,Y 530.946,Z 407.343,A -85,B 0,C 180,E1 -4522.573,E2 -4522.573} C_VEL
LIN {X 0,Y 530.964,Z 407.345,A -85,B 0,C 180,E1 -4525.06,E2 -4525.06} C_VEL
LIN {X 0,Y 531.011,Z 407.338,A -85,B 0,C 180,E1 -4527.596,E2 -4527.596} C_VEL
LIN {X 0,Y 530.962,Z 407.342,A -85,B 0,C 180,E1 -4529.91,E2 -4529.91} C_VEL
LIN {X 0,Y 530.301,Z 407.426,A -85,B 0,C 180,E1 -4530.543,E2 -4530.543} C_VEL
LIN {X 0,Y 527.432,Z 407.782,A -85,B 0,C 180,E1 -4531.57,E2 -4531.57} C_VEL
LIN {X 0,Y 525.018,Z 408.079,A -85,B 0,C 180,E1 -4532.398,E2 -4532.398} C_VEL
LIN {X 0,Y 524.006,Z 408.209,A -85,B 0,C 180,E1 -4533.037,E2 -4533.037} C_VEL
LIN {X 0,Y 523.936,Z 408.214,A -85,B 0,C 180,E1 -4533.253,E2 -4533.253} C_VEL
LIN {X 0,Y 523.903,Z 408.221,A -85,B 0,C 180,E1 -4536.175,E2 -4536.175} C_VEL
LIN {X 0,Y 523.924,Z 408.222,A -85,B 0,C 180,E1 -4539.085,E2 -4539.085} C_VEL
LIN {X 0,Y 523.955,Z 408.215,A -85,B 0,C 180,E1 -4542.119,E2 -4542.119} C_VEL
LIN {X 0,Y 523.957,Z 408.212,A -85,B 0,C 180,E1 -4545.309,E2 -4545.309} C_VEL
LIN {X 0,Y 523.959,Z 408.221,A -85,B 0,C 180,E1 -4548.69,E2 -4548.69} C_VEL
LIN {X 0,Y 523.919,Z 408.223,A -85,B 0,C 180,E1 -4551.081,E2 -4551.081} C_VEL
LIN {X 0,Y 523.898,Z 408.221,A -85,B 0,C 180,E1 -4553.825,E2 -4553.825} C_VEL
LIN {X 0,Y 523.944,Z 408.223,A -85,B 0,C 180,E1 -4556.636,E2 -4556.636} C_VEL
LIN {X 0,Y 523.947,Z 408.218,A -85,B 0,C 180,E1 -4559.355,E2 -4559.355} C_VEL
LIN {X 0,Y 523.92,Z 408.23,A -85,B 0,C 180,E1 -4562.294,E2 -4562.294} C_VEL
LIN {X 0,Y 523.953,Z 408.353,A -85,B 0,C 180,E1 -4565.506,E2 -4565.506} C_VEL
LIN {X 0,Y 525.485,Z 417.547,A -85,B 0,C 180,E1 -4566.971,E2 -4566.971} C_VEL
LIN {X 0,Y 525.09,Z 436.364,A -85,B 0,C 180,E1 -4569.84,E2 -4569.84} C_VEL
LIN {X 0,Y 524.67,Z 456.419,A -85,B 0,C 180,E1 -4572.861,E2 -4572.861} C_VEL
LIN {X 0,Y 524.454,Z 470.08,A -85,B 0,C 180,E1 -4574.889,E2 -4574.889} C_VEL
LIN {X 0,Y 525.904,Z 480.463,A -85,B 0,C 180,E1 -4575.081,E2 -4575.081} C_VEL
LIN {X 0,Y 525.513,Z 578.261,A -85,B 0,C 180,E1 -4576.44,E2 -4576.44} C_VEL
LIN {X 0,Y 525.294,Z 591.723,A -85,B 0,C 180,E1 -4576.779,E2 -4576.779} C_VEL
LIN {X 0,Y 525.061,Z 604.826,A -85,B 0,C 180,E1 -4577.29,E2 -4577.29} C_VEL
LIN {X 0,Y 524.813,Z 616.813,A -85,B 0,C 180,E1 -4577.922,E2 -4577.922} C_VEL
LIN {X 0,Y 524.591,Z 628.205,A -85,B 0,C 180,E1 -4578.701,E2 -4578.701} C_VEL
LIN {X 0,Y 524.236,Z 639.446,A -85,B 0,C 180,E1 -4579.671,E2 -4579.671} C_VEL
LIN {X 0,Y 524.002,Z 647.67,A -85,B 0,C 180,E1 -4580.543,E2 -4580.543} C_VEL
LIN {X 0,Y 523.826,Z 655.272,A -85,B 0,C 180,E1 -4581.513,E2 -4581.513} C_VEL
LIN {X 0,Y 523.629,Z 662.688,A -85,B 0,C 180,E1 -4582.674,E2 -4582.674} C_VEL
LIN {X 0,Y 523.541,Z 668.639,A -85,B 0,C 180,E1 -4583.835,E2 -4583.835} C_VEL
LIN {X 0,Y 523.383,Z 673.353,A -85,B 0,C 180,E1 -4584.993,E2 -4584.993} C_VEL
LIN {X 0,Y 523.443,Z 676.959,A -85,B 0,C 180,E1 -4586.151,E2 -4586.151} C_VEL
LIN {X 0,Y 523.367,Z 678.819,A -85,B 0,C 180,E1 -4586.921,E2 -4586.921} C_VEL
LIN {X 0,Y 523.335,Z 680.244,A -85,B 0,C 180,E1 -4587.691,E2 -4587.691} C_VEL
LIN {X 0,Y 523.25,Z 681.859,A -85,B 0,C 180,E1 -4589.23,E2 -4589.23} C_VEL
LIN {X 0,Y 523.247,Z 682.098,A -85,B 0,C 180,E1 -4590,E2 -4590} C_VEL
LIN {X 0,Y 523.25,Z 681.914,A -85,B 0,C 180,E1 -4590.77,E2 -4590.77} C_VEL
LIN {X 0,Y 523.335,Z 680.371,A -85,B 0,C 180,E1 -4592.309,E2 -4592.309} C_VEL
LIN {X 0,Y 523.368,Z 679.016,A -85,B 0,C 180,E1 -4593.079,E2 -4593.079} C_VEL
LIN {X 0,Y 523.442,Z 676.161,A -85,B 0,C 180,E1 -4594.235,E2 -4594.235} C_VEL
LIN {X 0,Y 523.462,Z 672.283,A -85,B 0,C 180,E1 -4595.393,E2 -4595.393} C_VEL
LIN {X 0,Y 523.556,Z 666.962,A -85,B 0,C 180,E1 -4596.611,E2 -4596.611} C_VEL
LIN {X 0,Y 523.72,Z 659.732,A -85,B 0,C 180,E1 -4597.906,E2 -4597.906} C_VEL
LIN {X 0,Y 523.879,Z 651.595,A -85,B 0,C 180,E1 -4599.069,E2 -4599.069} C_VEL
LIN {X 0,Y 524.099,Z 643.215,A -85,B 0,C 180,E1 -4600.039,E2 -4600.039} C_VEL
LIN {X 0,Y 524.438,Z 632.93,A -85,B 0,C 180,E1 -4601.009,E2 -4601.009} C_VEL
LIN {X 0,Y 524.713,Z 622.702,A -85,B 0,C 180,E1 -4601.79,E2 -4601.79} C_VEL
LIN {X 0,Y 524.967,Z 611.543,A -85,B 0,C 180,E1 -4602.467,E2 -4602.467} C_VEL
LIN {X 0,Y 525.231,Z 598.933,A -85,B 0,C 180,E1 -4603.05,E2 -4603.05} C_VEL
LIN {X 0,Y 525.437,Z 586.486,A -85,B 0,C 180,E1 -4603.463,E2 -4603.463} C_VEL
LIN {X 0,Y 525.59,Z 573.558,A -85,B 0,C 180,E1 -4603.73,E2 -4603.73} C_VEL
LIN {X 0,Y 525.824,Z 478.383,A -85,B 0,C 180,E1 -4605.041,E2 -4605.041} C_VEL
LIN {X 0,Y 524.463,Z 469.957,A -85,B 0,C 180,E1 -4605.199,E2 -4605.199} C_VEL
LIN {X 0,Y 524.809,Z 449.288,A -85,B 0,C 180,E1 -4608.302,E2 -4608.302} C_VEL
LIN {X 0,Y 525.197,Z 430.263,A -85,B 0,C 180,E1 -4611.18,E2 -4611.18} C_VEL
LIN {X 0,Y 525.458,Z 416.761,A -85,B 0,C 180,E1 -4613.239,E2 -4613.239} C_VEL
LIN {X 0,Y 523.929,Z 408.223,A -85,B 0,C 180,E1 -4614.625,E2 -4614.625} C_VEL
LIN {X 0,Y 523.92,Z 408.228,A -85,B 0,C 180,E1 -4617.706,E2 -4617.706} C_VEL
LIN {X 0,Y 523.947,Z 408.217,A -85,B 0,C 180,E1 -4620.645,E2 -4620.645} C_VEL
LIN {X 0,Y 523.962,Z 408.221,A -85,B 0,C 180,E1 -4623.734,E2 -4623.734} C_VEL
LIN {X 0,Y 523.901,Z 408.223,A -85,B 0,C 180,E1 -4626.401,E2 -4626.401} C_VEL
LIN {X 0,Y 523.922,Z 408.225,A -85,B 0,C 180,E1 -4629.085,E2 -4629.085} C_VEL
LIN {X 0,Y 523.955,Z 408.215,A -85,B 0,C 180,E1 -4632.119,E2 -4632.119} C_VEL
LIN {X 0,Y 523.96,Z 408.22,A -85,B 0,C 180,E1 -4635.309,E2 -4635.309} C_VEL
LIN {X 0,Y 523.959,Z 408.217,A -85,B 0,C 180,E1 -4638.69,E2 -4638.69} C_VEL
LIN {X 0,Y 523.921,Z 408.224,A -85,B 0,C 180,E1 -4641.08,E2 -4641.08} C_VEL
LIN {X 0,Y 523.898,Z 408.217,A -85,B 0,C 180,E1 -4643.825,E2 -4643.825} C_VEL
LIN {X 0,Y 523.945,Z 408.224,A -85,B 0,C 180,E1 -4646.636,E2 -4646.636} C_VEL
LIN {X 0,Y 523.947,Z 408.216,A -85,B 0,C 180,E1 -4649.355,E2 -4649.355} C_VEL
LIN {X 0,Y 523.923,Z 408.226,A -85,B 0,C 180,E1 -4652.294,E2 -4652.294} C_VEL
LIN {X 0,Y 523.971,Z 408.387,A -85,B 0,C 180,E1 -4655.508,E2 -4655.508} C_VEL
LIN {X 0,Y 525.4,Z 416.194,A -85,B 0,C 180,E1 -4656.758,E2 -4656.758} C_VEL
LIN {X 0,Y 525.195,Z 432.509,A -85,B 0,C 180,E1 -4659.23,E2 -4659.23} C_VEL
LIN {X 0,Y 524.78,Z 452.565,A -85,B 0,C 180,E1 -4662.261,E2 -4662.261} C_VEL
LIN {X 0,Y 524.414,Z 470.046,A -85,B 0,C 180,E1 -4664.905,E2 -4664.905} C_VEL
LIN {X 0,Y 525.852,Z 479.022,A -85,B 0,C 180,E1 -4665.082,E2 -4665.082} C_VEL
LIN {X 0,Y 525.454,Z 575.87,A -85,B 0,C 180,E1 -4666.439,E2 -4666.439} C_VEL
LIN {X 0,Y 525.296,Z 587.722,A -85,B 0,C 180,E1 -4666.706,E2 -4666.706} C_VEL
LIN {X 0,Y 525.083,Z 600.565,A -85,B 0,C 180,E1 -4667.143,E2 -4667.143} C_VEL
LIN {X 0,Y 524.827,Z 613.093,A -85,B 0,C 180,E1 -4667.746,E2 -4667.746} C_VEL
LIN {X 0,Y 524.639,Z 623.646,A -85,B 0,C 180,E1 -4668.408,E2 -4668.408} C_VEL
LIN {X 0,Y 524.401,Z 632.547,A -85,B 0,C 180,E1 -4669.088,E2 -4669.088} C_VEL
LIN {X 0,Y 524.188,Z 640.055,A -85,B 0,C 180,E1 -4669.767,E2 -4669.767} C_VEL
LIN {X 0,Y 523.989,Z 647.356,A -85,B 0,C 180,E1 -4670.543,E2 -4670.543} C_VEL
LIN {X 0,Y 523.797,Z 655.01,A -85,B 0,C 180,E1 -4671.513,E2 -4671.513} C_VEL
LIN {X 0,Y 523.637,Z 661.367,A -85,B 0,C 180,E1 -4672.481,E2 -4672.481} C_VEL
LIN {X 0,Y 523.526,Z 666.506,A -85,B 0,C 180,E1 -4673.417,E2 -4673.417} C_VEL
LIN {X 0,Y 523.54,Z 670.247,A -85,B 0,C 180,E1 -4674.222,E2 -4674.222} C_VEL
LIN {X 0,Y 523.369,Z 674.591,A -85,B 0,C 180,E1 -4675.379,E2 -4675.379} C_VEL
LIN {X 0,Y 523.444,Z 676.957,A -85,B 0,C 180,E1 -4676.151,E2 -4676.151} C_VEL
LIN {X 0,Y 523.367,Z 678.771,A -85,B 0,C 180,E1 -4676.921,E2 -4676.921} C_VEL
LIN {X 0,Y 523.274,Z 681.249,A -85,B 0,C 180,E1 -4678.461,E2 -4678.461} C_VEL
LIN {X 0,Y 523.25,Z 681.841,A -85,B 0,C 180,E1 -4679.23,E2 -4679.23} C_VEL
LIN {X 0,Y 523.25,Z 681.908,A -85,B 0,C 180,E1 -4680.77,E2 -4680.77} C_VEL
LIN {X 0,Y 523.275,Z 681.325,A -85,B 0,C 180,E1 -4681.539,E2 -4681.539} C_VEL
LIN {X 0,Y 523.368,Z 678.984,A -85,B 0,C 180,E1 -4683.079,E2 -4683.079} C_VEL
LIN {X 0,Y 523.441,Z 676.103,A -85,B 0,C 180,E1 -4684.235,E2 -4684.235} C_VEL
LIN {X 0,Y 523.463,Z 672.186,A -85,B 0,C 180,E1 -4685.393,E2 -4685.393} C_VEL
LIN {X 0,Y 523.517,Z 667.012,A -85,B 0,C 180,E1 -4686.575,E2 -4686.575} C_VEL
LIN {X 0,Y 523.626,Z 661.929,A -85,B 0,C 180,E1 -4687.519,E2 -4687.519} C_VEL
LIN {X 0,Y 523.811,Z 655.669,A -85,B 0,C 180,E1 -4688.487,E2 -4688.487} C_VEL
LIN {X 0,Y 523.964,Z 648.128,A -85,B 0,C 180,E1 -4689.457,E2 -4689.457} C_VEL
LIN {X 0,Y 524.218,Z 639,A -85,B 0,C 180,E1 -4690.427,E2 -4690.427} C_VEL
LIN {X 0,Y 524.526,Z 627.578,A -85,B 0,C 180,E1 -4691.399,E2 -4691.399} C_VEL
LIN {X 0,Y 524.77,Z 616.589,A -85,B 0,C 180,E1 -4692.134,E2 -4692.134} C_VEL
LIN {X 0,Y 524.952,Z 605.666,A -85,B 0,C 180,E1 -4692.713,E2 -4692.713} C_VEL
LIN {X 0,Y 525.242,Z 592.863,A -85,B 0,C 180,E1 -4693.222,E2 -4693.222} C_VEL
LIN {X 0,Y 525.41,Z 580.182,A -85,B 0,C 180,E1 -4693.562,E2 -4693.562} C_VEL
LIN {X 0,Y 525.58,Z 548.579,A -85,B 0,C 180,E1 -4694.026,E2 -4694.026} C_VEL
LIN {X 0,Y 525.857,Z 479.024,A -85,B 0,C 180,E1 -4695.006,E2 -4695.006} C_VEL
LIN {X 0,Y 524.443,Z 470.048,A -85,B 0,C 180,E1 -4695.194,E2 -4695.194} C_VEL
LIN {X 0,Y 524.713,Z 455.778,A -85,B 0,C 180,E1 -4697.339,E2 -4697.339} C_VEL
LIN {X 0,Y 525.077,Z 434.668,A -85,B 0,C 180,E1 -4700.457,E2 -4700.457} C_VEL
LIN {X 0,Y 525.273,Z 416.835,A -85,B 0,C 180,E1 -4703.039,E2 -4703.039} C_VEL
LIN {X 0,Y 524.373,Z 410.69,A -85,B 0,C 180,E1 -4703.958,E2 -4703.958} C_VEL
LIN {X 0,Y 523.93,Z 408.225,A -85,B 0,C 180,E1 -4704.344,E2 -4704.344} C_VEL
LIN {X 0,Y 523.9,Z 408.226,A -85,B 0,C 180,E1 -4707.136,E2 -4707.136} C_VEL
LIN {X 0,Y 523.899,Z 408.23,A -85,B 0,C 180,E1 -4709.759,E2 -4709.759} C_VEL
LIN {X 0,Y 523.936,Z 408.219,A -85,B 0,C 180,E1 -4712.449,E2 -4712.449} C_VEL
LIN {X 0,Y 523.921,Z 408.226,A -85,B 0,C 180,E1 -4715.227,E2 -4715.227} C_VEL
LIN {X 0,Y 523.916,Z 408.22,A -85,B 0,C 180,E1 -4718.102,E2 -4718.102} C_VEL
LIN {X 0,Y 523.942,Z 408.223,A -85,B 0,C 180,E1 -4721.092,E2 -4721.092} C_VEL
LIN {X 0,Y 523.945,Z 408.217,A -85,B 0,C 180,E1 -4724.228,E2 -4724.228} C_VEL
LIN {X 0,Y 523.925,Z 408.225,A -85,B 0,C 180,E1 -4726.833,E2 -4726.833} C_VEL
LIN {X 0,Y 523.94,Z 408.217,A -85,B 0,C 180,E1 -4729.87,E2 -4729.87} C_VEL
LIN {X 0,Y 523.907,Z 408.227,A -85,B 0,C 180,E1 -4732.868,E2 -4732.868} C_VEL
LIN {X 0,Y 523.934,Z 408.218,A -85,B 0,C 180,E1 -4735.71,E2 -4735.71} C_VEL
LIN {X 0,Y 523.921,Z 408.226,A -85,B 0,C 180,E1 -4738.456,E2 -4738.456} C_VEL
LIN {X 0,Y 523.91,Z 408.224,A -85,B 0,C 180,E1 -4741.123,E2 -4741.123} C_VEL
LIN {X 0,Y 523.962,Z 408.418,A -85,B 0,C 180,E1 -4742.956,E2 -4742.956} C_VEL
LIN {X 0,Y 526.093,Z 418.803,A -85,B 0,C 180,E1 -4744.48,E2 -4744.48} C_VEL
LIN {X 0,Y 525.691,Z 437.383,A -85,B 0,C 180,E1 -4746.98,E2 -4746.98} C_VEL
LIN {X 0,Y 525.256,Z 456.306,A -85,B 0,C 180,E1 -4749.49,E2 -4749.49} C_VEL
LIN {X 0,Y 524.814,Z 479.054,A -85,B 0,C 180,E1 -4752.464,E2 -4752.464} C_VEL
LIN {X 0,Y 524.465,Z 497.392,A -85,B 0,C 180,E1 -4754.84,E2 -4754.84} C_VEL
LIN {X 0,Y 525.855,Z 509.615,A -85,B 0,C 180,E1 -4755.065,E2 -4755.065} C_VEL
LIN {X 0,Y 525.46,Z 604.959,A -85,B 0,C 180,E1 -4756.39,E2 -4756.39} C_VEL
LIN {X 0,Y 525.249,Z 618.336,A -85,B 0,C 180,E1 -4756.704,E2 -4756.704} C_VEL
LIN {X 0,Y 524.995,Z 631.63,A -85,B 0,C 180,E1 -4757.19,E2 -4757.19} C_VEL
LIN {X 0,Y 524.76,Z 644.218,A -85,B 0,C 180,E1 -4757.824,E2 -4757.824} C_VEL
LIN {X 0,Y 524.491,Z 656.043,A -85,B 0,C 180,E1 -4758.601,E2 -4758.601} C_VEL
LIN {X 0,Y 524.201,Z 666.653,A -85,B 0,C 180,E1 -4759.475,E2 -4759.475} C_VEL
LIN {X 0,Y 524.005,Z 675.336,A -85,B 0,C 180,E1 -4760.349,E2 -4760.349} C_VEL
LIN {X 0,Y 523.806,Z 683.355,A -85,B 0,C 180,E1 -4761.318,E2 -4761.318} C_VEL
LIN {X 0,Y 523.617,Z 691.177,A -85,B 0,C 180,E1 -4762.48,E2 -4762.48} C_VEL
LIN {X 0,Y 523.522,Z 696.388,A -85,B 0,C 180,E1 -4763.42,E2 -4763.42} C_VEL
LIN {X 0,Y 523.464,Z 701.727,A -85,B 0,C 180,E1 -4764.607,E2 -4764.607} C_VEL
LIN {X 0,Y 523.425,Z 705.756,A -85,B 0,C 180,E1 -4765.765,E2 -4765.765} C_VEL
LIN {X 0,Y 523.367,Z 708.727,A -85,B 0,C 180,E1 -4766.921,E2 -4766.921} C_VEL
LIN {X 0,Y 523.335,Z 710.136,A -85,B 0,C 180,E1 -4767.691,E2 -4767.691} C_VEL
LIN {X 0,Y 523.25,Z 711.747,A -85,B 0,C 180,E1 -4769.23,E2 -4769.23} C_VEL
LIN {X 0,Y 523.246,Z 711.964,A -85,B 0,C 180,E1 -4770,E2 -4770} C_VEL
LIN {X 0,Y 523.274,Z 711.138,A -85,B 0,C 180,E1 -4771.539,E2 -4771.539} C_VEL
LIN {X 0,Y 523.335,Z 710.139,A -85,B 0,C 180,E1 -4772.309,E2 -4772.309} C_VEL
LIN {X 0,Y 523.367,Z 708.73,A -85,B 0,C 180,E1 -4773.079,E2 -4773.079} C_VEL
LIN {X 0,Y 523.425,Z 705.755,A -85,B 0,C 180,E1 -4774.235,E2 -4774.235} C_VEL
LIN {X 0,Y 523.464,Z 701.715,A -85,B 0,C 180,E1 -4775.393,E2 -4775.393} C_VEL
LIN {X 0,Y 523.523,Z 696.353,A -85,B 0,C 180,E1 -4776.581,E2 -4776.581} C_VEL
LIN {X 0,Y 523.665,Z 689.942,A -85,B 0,C 180,E1 -4777.713,E2 -4777.713} C_VEL
LIN {X 0,Y 523.845,Z 681.757,A -85,B 0,C 180,E1 -4778.875,E2 -4778.875} C_VEL
LIN {X 0,Y 524.054,Z 673.408,A -85,B 0,C 180,E1 -4779.845,E2 -4779.845} C_VEL
LIN {X 0,Y 524.307,Z 663.197,A -85,B 0,C 180,E1 -4780.816,E2 -4780.816} C_VEL
LIN {X 0,Y 524.6,Z 651.678,A -85,B 0,C 180,E1 -4781.689,E2 -4781.689} C_VEL
LIN {X 0,Y 524.807,Z 640.306,A -85,B 0,C 180,E1 -4782.372,E2 -4782.372} C_VEL
LIN {X 0,Y 525.054,Z 627.629,A -85,B 0,C 180,E1 -4782.956,E2 -4782.956} C_VEL
LIN {X 0,Y 525.283,Z 614.106,A -85,B 0,C 180,E1 -4783.393,E2 -4783.393} C_VEL
LIN {X 0,Y 525.478,Z 600.882,A -85,B 0,C 180,E1 -4783.659,E2 -4783.659} C_VEL
LIN {X 0,Y 525.772,Z 507.642,A -85,B 0,C 180,E1 -4784.948,E2 -4784.948} C_VEL
LIN {X 0,Y 524.413,Z 496.672,A -85,B 0,C 180,E1 -4785.16,E2 -4785.16} C_VEL
LIN {X 0,Y 524.805,Z 472.041,A -85,B 0,C 180,E1 -4788.303,E2 -4788.303} C_VEL
LIN {X 0,Y 525.271,Z 448.109,A -85,B 0,C 180,E1 -4791.383,E2 -4791.383} C_VEL
LIN {X 0,Y 525.686,Z 424.406,A -85,B 0,C 180,E1 -4794.485,E2 -4794.485} C_VEL
LIN {X 0,Y 525.584,Z 416.482,A -85,B 0,C 180,E1 -4795.546,E2 -4795.546} C_VEL
LIN {X 0,Y 523.945,Z 408.221,A -85,B 0,C 180,E1 -4796.756,E2 -4796.756} C_VEL
LIN {X 0,Y 523.899,Z 408.231,A -85,B 0,C 180,E1 -4799.759,E2 -4799.759} C_VEL
LIN {X 0,Y 523.935,Z 408.219,A -85,B 0,C 180,E1 -4802.45,E2 -4802.45} C_VEL
LIN {X 0,Y 523.919,Z 408.225,A -85,B 0,C 180,E1 -4805.227,E2 -4805.227} C_VEL
LIN {X 0,Y 523.915,Z 408.221,A -85,B 0,C 180,E1 -4808.102,E2 -4808.102} C_VEL
LIN {X 0,Y 523.94,Z 408.223,A -85,B 0,C 180,E1 -4811.093,E2 -4811.093} C_VEL
LIN {X 0,Y 523.934,Z 408.218,A -85,B 0,C 180,E1 -4814.229,E2 -4814.229} C_VEL
LIN {X 0,Y 523.92,Z 408.223,A -85,B 0,C 180,E1 -4816.833,E2 -4816.833} C_VEL
LIN {X 0,Y 523.942,Z 408.221,A -85,B 0,C 180,E1 -4818.908,E2 -4818.908} C_VEL
LIN {X 0,Y 523.918,Z 408.22,A -85,B 0,C 180,E1 -4821.898,E2 -4821.898} C_VEL
LIN {X 0,Y 523.931,Z 408.224,A -85,B 0,C 180,E1 -4824.911,E2 -4824.911} C_VEL
LIN {X 0,Y 523.938,Z 408.218,A -85,B 0,C 180,E1 -4827.68,E2 -4827.68} C_VEL
LIN {X 0,Y 523.956,Z 408.221,A -85,B 0,C 180,E1 -4830.677,E2 -4830.677} C_VEL
LIN {X 0,Y 523.975,Z 408.214,A -85,B 0,C 180,E1 -4833.729,E2 -4833.729} C_VEL
LIN {X 0,Y 523.917,Z 408.225,A -85,B 0,C 180,E1 -4836.27,E2 -4836.27} C_VEL
LIN {X 0,Y 523.948,Z 408.224,A -85,B 0,C 180,E1 -4838.767,E2 -4838.767} C_VEL
LIN {X 0,Y 523.941,Z 408.22,A -85,B 0,C 180,E1 -4841.22,E2 -4841.22} C_VEL
LIN {X 0,Y 523.912,Z 408.223,A -85,B 0,C 180,E1 -4843.638,E2 -4843.638} C_VEL
LIN {X 0,Y 523.982,Z 408.219,A -85,B 0,C 180,E1 -4844.974,E2 -4844.974} C_VEL
LIN {X 0,Y 525.991,Z 414.877,A -85,B 0,C 180,E1 -4845.138,E2 -4845.138} C_VEL
LIN {X 0,Y 525.466,Z 510.378,A -85,B 0,C 180,E1 -4846.513,E2 -4846.513} C_VEL
LIN {X 0,Y 525.286,Z 524.342,A -85,B 0,C 180,E1 -4846.878,E2 -4846.878} C_VEL
LIN {X 0,Y 525.091,Z 536.164,A -85,B 0,C 180,E1 -4847.34,E2 -4847.34} C_VEL
LIN {X 0,Y 524.86,Z 548.161,A -85,B 0,C 180,E1 -4847.97,E2 -4847.97} C_VEL
LIN {X 0,Y 524.564,Z 560.264,A -85,B 0,C 180,E1 -4848.798,E2 -4848.798} C_VEL
LIN {X 0,Y 524.366,Z 569.328,A -85,B 0,C 180,E1 -4849.576,E2 -4849.576} C_VEL
LIN {X 0,Y 524.1,Z 578.574,A -85,B 0,C 180,E1 -4850.545,E2 -4850.545} C_VEL
LIN {X 0,Y 523.926,Z 586.189,A -85,B 0,C 180,E1 -4851.515,E2 -4851.515} C_VEL
LIN {X 0,Y 523.703,Z 593.651,A -85,B 0,C 180,E1 -4852.676,E2 -4852.676} C_VEL
LIN {X 0,Y 523.588,Z 599.587,A -85,B 0,C 180,E1 -4853.836,E2 -4853.836} C_VEL
LIN {X 0,Y 523.451,Z 604.25,A -85,B 0,C 180,E1 -4854.993,E2 -4854.993} C_VEL
LIN {X 0,Y 523.476,Z 607.809,A -85,B 0,C 180,E1 -4856.151,E2 -4856.151} C_VEL
LIN {X 0,Y 523.428,Z 609.679,A -85,B 0,C 180,E1 -4856.921,E2 -4856.921} C_VEL
LIN {X 0,Y 523.35,Z 611.091,A -85,B 0,C 180,E1 -4857.691,E2 -4857.691} C_VEL
LIN {X 0,Y 523.282,Z 612.672,A -85,B 0,C 180,E1 -4859.23,E2 -4859.23} C_VEL
LIN {X 0,Y 523.28,Z 612.913,A -85,B 0,C 180,E1 -4860,E2 -4860} C_VEL
LIN {X 0,Y 523.296,Z 612.108,A -85,B 0,C 180,E1 -4861.539,E2 -4861.539} C_VEL
LIN {X 0,Y 523.346,Z 611.184,A -85,B 0,C 180,E1 -4862.309,E2 -4862.309} C_VEL
LIN {X 0,Y 523.424,Z 609.785,A -85,B 0,C 180,E1 -4863.079,E2 -4863.079} C_VEL
LIN {X 0,Y 523.48,Z 606.946,A -85,B 0,C 180,E1 -4864.235,E2 -4864.235} C_VEL
LIN {X 0,Y 523.476,Z 603.087,A -85,B 0,C 180,E1 -4865.393,E2 -4865.393} C_VEL
LIN {X 0,Y 523.6,Z 597.541,A -85,B 0,C 180,E1 -4866.653,E2 -4866.653} C_VEL
LIN {X 0,Y 523.746,Z 591.701,A -85,B 0,C 180,E1 -4867.712,E2 -4867.712} C_VEL
LIN {X 0,Y 523.912,Z 585.242,A -85,B 0,C 180,E1 -4868.68,E2 -4868.68} C_VEL
LIN {X 0,Y 524.098,Z 577.463,A -85,B 0,C 180,E1 -4869.65,E2 -4869.65} C_VEL
LIN {X 0,Y 524.377,Z 567.996,A -85,B 0,C 180,E1 -4870.62,E2 -4870.62} C_VEL
LIN {X 0,Y 524.638,Z 557.37,A -85,B 0,C 180,E1 -4871.494,E2 -4871.494} C_VEL
LIN {X 0,Y 524.886,Z 546.706,A -85,B 0,C 180,E1 -4872.193,E2 -4872.193} C_VEL
LIN {X 0,Y 525.069,Z 534.792,A -85,B 0,C 180,E1 -4872.808,E2 -4872.808} C_VEL
LIN {X 0,Y 525.344,Z 521.067,A -85,B 0,C 180,E1 -4873.318,E2 -4873.318} C_VEL
LIN {X 0,Y 525.455,Z 508.939,A -85,B 0,C 180,E1 -4873.61,E2 -4873.61} C_VEL
LIN {X 0,Y 525.82,Z 414.11,A -85,B 0,C 180,E1 -4874.962,E2 -4874.962} C_VEL
LIN {X 0,Y 523.961,Z 408.22,A -85,B 0,C 180,E1 -4875.112,E2 -4875.112} C_VEL
LIN {X 0,Y 523.919,Z 408.224,A -85,B 0,C 180,E1 -4877.971,E2 -4877.971} C_VEL
LIN {X 0,Y 523.961,Z 408.216,A -85,B 0,C 180,E1 -4880.411,E2 -4880.411} C_VEL
LIN {X 0,Y 523.912,Z 408.221,A -85,B 0,C 180,E1 -4882.894,E2 -4882.894} C_VEL
LIN {X 0,Y 523.912,Z 408.227,A -85,B 0,C 180,E1 -4885.421,E2 -4885.421} C_VEL
LIN {X 0,Y 523.959,Z 408.213,A -85,B 0,C 180,E1 -4888,E2 -4888} C_VEL
LIN {X 0,Y 523.948,Z 408.219,A -85,B 0,C 180,E1 -4890.855,E2 -4890.855} C_VEL
LIN {X 0,Y 523.936,Z 408.214,A -85,B 0,C 180,E1 -4893.253,E2 -4893.253} C_VEL
LIN {X 0,Y 523.293,Z 408.297,A -85,B 0,C 180,E1 -4893.895,E2 -4893.895} C_VEL
LIN {X 0,Y 520.409,Z 408.656,A -85,B 0,C 180,E1 -4894.936,E2 -4894.936} C_VEL
LIN {X 0,Y 517.97,Z 408.961,A -85,B 0,C 180,E1 -4895.775,E2 -4895.775} C_VEL
LIN {X 0,Y 516.947,Z 409.089,A -85,B 0,C 180,E1 -4896.424,E2 -4896.424} C_VEL
LIN {X 0,Y 516.879,Z 409.099,A -85,B 0,C 180,E1 -4896.643,E2 -4896.643} C_VEL
LIN {X 0,Y 516.885,Z 409.092,A -85,B 0,C 180,E1 -4899.721,E2 -4899.721} C_VEL
LIN {X 0,Y 516.915,Z 409.091,A -85,B 0,C 180,E1 -4901.775,E2 -4901.775} C_VEL
LIN {X 0,Y 516.926,Z 409.091,A -85,B 0,C 180,E1 -4905.01,E2 -4905.01} C_VEL
LIN {X 0,Y 516.916,Z 409.096,A -85,B 0,C 180,E1 -4908.399,E2 -4908.399} C_VEL
LIN {X 0,Y 516.882,Z 409.098,A -85,B 0,C 180,E1 -4911.284,E2 -4911.284} C_VEL
LIN {X 0,Y 516.87,Z 409.1,A -85,B 0,C 180,E1 -4914.219,E2 -4914.219} C_VEL
LIN {X 0,Y 516.898,Z 409.096,A -85,B 0,C 180,E1 -4917.053,E2 -4917.053} C_VEL
LIN {X 0,Y 516.87,Z 409.101,A -85,B 0,C 180,E1 -4919.795,E2 -4919.795} C_VEL
LIN {X 0,Y 516.876,Z 409.106,A -85,B 0,C 180,E1 -4922.464,E2 -4922.464} C_VEL
LIN {X 0,Y 516.931,Z 409.273,A -85,B 0,C 180,E1 -4925.339,E2 -4925.339} C_VEL
LIN {X 0,Y 518.547,Z 418.683,A -85,B 0,C 180,E1 -4926.856,E2 -4926.856} C_VEL
LIN {X 0,Y 518.131,Z 437.576,A -85,B 0,C 180,E1 -4929.773,E2 -4929.773} C_VEL
LIN {X 0,Y 517.696,Z 457.688,A -85,B 0,C 180,E1 -4932.826,E2 -4932.826} C_VEL
LIN {X 0,Y 517.48,Z 470.257,A -85,B 0,C 180,E1 -4934.679,E2 -4934.679} C_VEL
LIN {X 0,Y 519.064,Z 480.667,A -85,B 0,C 180,E1 -4934.881,E2 -4934.881} C_VEL
LIN {X 0,Y 518.626,Z 578.368,A -85,B 0,C 180,E1 -4936.257,E2 -4936.257} C_VEL
LIN {X 0,Y 518.392,Z 591.868,A -85,B 0,C 180,E1 -4936.6,E2 -4936.6} C_VEL
LIN {X 0,Y 518.147,Z 604.99,A -85,B 0,C 180,E1 -4937.117,E2 -4937.117} C_VEL
LIN {X 0,Y 517.877,Z 616.271,A -85,B 0,C 180,E1 -4937.715,E2 -4937.715} C_VEL
LIN {X 0,Y 517.677,Z 627.128,A -85,B 0,C 180,E1 -4938.449,E2 -4938.449} C_VEL
LIN {X 0,Y 517.306,Z 637.572,A -85,B 0,C 180,E1 -4939.333,E2 -4939.333} C_VEL
LIN {X 0,Y 516.992,Z 647.856,A -85,B 0,C 180,E1 -4940.414,E2 -4940.414} C_VEL
LIN {X 0,Y 516.747,Z 656.789,A -85,B 0,C 180,E1 -4941.593,E2 -4941.593} C_VEL
LIN {X 0,Y 516.561,Z 663.96,A -85,B 0,C 180,E1 -4942.77,E2 -4942.77} C_VEL
LIN {X 0,Y 516.467,Z 668.829,A -85,B 0,C 180,E1 -4943.75,E2 -4943.75} C_VEL
LIN {X 0,Y 516.313,Z 673.543,A -85,B 0,C 180,E1 -4944.924,E2 -4944.924} C_VEL
LIN {X 0,Y 516.373,Z 677.149,A -85,B 0,C 180,E1 -4946.098,E2 -4946.098} C_VEL
LIN {X 0,Y 516.282,Z 679.009,A -85,B 0,C 180,E1 -4946.879,E2 -4946.879} C_VEL
LIN {X 0,Y 516.261,Z 680.433,A -85,B 0,C 180,E1 -4947.659,E2 -4947.659} C_VEL
LIN {X 0,Y 516.16,Z 682.048,A -85,B 0,C 180,E1 -4949.22,E2 -4949.22} C_VEL
LIN {X 0,Y 516.155,Z 682.287,A -85,B 0,C 180,E1 -4950,E2 -4950} C_VEL
LIN {X 0,Y 516.16,Z 682.102,A -85,B 0,C 180,E1 -4950.78,E2 -4950.78} C_VEL
LIN {X 0,Y 516.261,Z 680.558,A -85,B 0,C 180,E1 -4952.341,E2 -4952.341} C_VEL
LIN {X 0,Y 516.283,Z 679.203,A -85,B 0,C 180,E1 -4953.121,E2 -4953.121} C_VEL
LIN {X 0,Y 516.362,Z 676.347,A -85,B 0,C 180,E1 -4954.293,E2 -4954.293} C_VEL
LIN {X 0,Y 516.403,Z 672.468,A -85,B 0,C 180,E1 -4955.467,E2 -4955.467} C_VEL
LIN {X 0,Y 516.502,Z 666.528,A -85,B 0,C 180,E1 -4956.825,E2 -4956.825} C_VEL
LIN {X 0,Y 516.665,Z 659.913,A -85,B 0,C 180,E1 -4958.015,E2 -4958.015} C_VEL
LIN {X 0,Y 516.856,Z 651.772,A -85,B 0,C 180,E1 -4959.194,E2 -4959.194} C_VEL
LIN {X 0,Y 517.095,Z 643.388,A -85,B 0,C 180,E1 -4960.177,E2 -4960.177} C_VEL
LIN {X 0,Y 517.467,Z 633.096,A -85,B 0,C 180,E1 -4961.159,E2 -4961.159} C_VEL
LIN {X 0,Y 517.755,Z 623.097,A -85,B 0,C 180,E1 -4961.934,E2 -4961.934} C_VEL
LIN {X 0,Y 518.036,Z 611.688,A -85,B 0,C 180,E1 -4962.636,E2 -4962.636} C_VEL
LIN {X 0,Y 518.312,Z 599.06,A -85,B 0,C 180,E1 -4963.227,E2 -4963.227} C_VEL
LIN {X 0,Y 518.547,Z 586.572,A -85,B 0,C 180,E1 -4963.645,E2 -4963.645} C_VEL
LIN {X 0,Y 518.703,Z 573.559,A -85,B 0,C 180,E1 -4963.916,E2 -4963.916} C_VEL
LIN {X 0,Y 519.018,Z 479.497,A -85,B 0,C 180,E1 -4965.227,E2 -4965.227} C_VEL
LIN {X 0,Y 517.475,Z 469.928,A -85,B 0,C 180,E1 -4965.425,E2 -4965.425} C_VEL
LIN {X 0,Y 517.886,Z 448.888,A -85,B 0,C 180,E1 -4968.597,E2 -4968.597} C_VEL
LIN {X 0,Y 518.253,Z 431.406,A -85,B 0,C 180,E1 -4971.27,E2 -4971.27} C_VEL
LIN {X 0,Y 518.493,Z 417.875,A -85,B 0,C 180,E1 -4973.358,E2 -4973.358} C_VEL
LIN {X 0,Y 516.876,Z 409.102,A -85,B 0,C 180,E1 -4974.82,E2 -4974.82} C_VEL
LIN {X 0,Y 516.868,Z 409.105,A -85,B 0,C 180,E1 -4977.892,E2 -4977.892} C_VEL
LIN {X 0,Y 516.87,Z 409.1,A -85,B 0,C 180,E1 -4980.205,E2 -4980.205} C_VEL
LIN {X 0,Y 516.898,Z 409.098,A -85,B 0,C 180,E1 -4982.947,E2 -4982.947} C_VEL
LIN {X 0,Y 516.871,Z 409.102,A -85,B 0,C 180,E1 -4985.781,E2 -4985.781} C_VEL
LIN {X 0,Y 516.882,Z 409.098,A -85,B 0,C 180,E1 -4988.716,E2 -4988.716} C_VEL
LIN {X 0,Y 516.915,Z 409.094,A -85,B 0,C 180,E1 -4991.775,E2 -4991.775} C_VEL
LIN {X 0,Y 516.926,Z 409.097,A -85,B 0,C 180,E1 -4995.01,E2 -4995.01} C_VEL
LIN {X 0,Y 516.917,Z 409.091,A -85,B 0,C 180,E1 -4998.399,E2 -4998.399} C_VEL
LIN {X 0,Y 516.884,Z 409.098,A -85,B 0,C 180,E1 -5001.284,E2 -5001.284} C_VEL
LIN {X 0,Y 516.871,Z 409.094,A -85,B 0,C 180,E1 -5004.219,E2 -5004.219} C_VEL
LIN {X 0,Y 516.898,Z 409.097,A -85,B 0,C 180,E1 -5007.053,E2 -5007.053} C_VEL
LIN {X 0,Y 516.87,Z 409.099,A -85,B 0,C 180,E1 -5009.795,E2 -5009.795} C_VEL
LIN {X 0,Y 516.879,Z 409.103,A -85,B 0,C 180,E1 -5012.464,E2 -5012.464} C_VEL
LIN {X 0,Y 516.931,Z 409.293,A -85,B 0,C 180,E1 -5015.339,E2 -5015.339} C_VEL
LIN {X 0,Y 518.54,Z 418.698,A -85,B 0,C 180,E1 -5016.855,E2 -5016.855} C_VEL
LIN {X 0,Y 518.156,Z 437.763,A -85,B 0,C 180,E1 -5019.771,E2 -5019.771} C_VEL
LIN {X 0,Y 517.71,Z 457.89,A -85,B 0,C 180,E1 -5022.827,E2 -5022.827} C_VEL
LIN {X 0,Y 517.471,Z 470.308,A -85,B 0,C 180,E1 -5024.704,E2 -5024.704} C_VEL
LIN {X 0,Y 519.013,Z 480.589,A -85,B 0,C 180,E1 -5024.905,E2 -5024.905} C_VEL
LIN {X 0,Y 518.541,Z 577.755,A -85,B 0,C 180,E1 -5026.304,E2 -5026.304} C_VEL
LIN {X 0,Y 518.315,Z 590.716,A -85,B 0,C 180,E1 -5026.623,E2 -5026.623} C_VEL
LIN {X 0,Y 518.086,Z 604.733,A -85,B 0,C 180,E1 -5027.166,E2 -5027.166} C_VEL
LIN {X 0,Y 517.812,Z 615.792,A -85,B 0,C 180,E1 -5027.748,E2 -5027.748} C_VEL
LIN {X 0,Y 517.595,Z 626.31,A -85,B 0,C 180,E1 -5028.447,E2 -5028.447} C_VEL
LIN {X 0,Y 517.3,Z 637.022,A -85,B 0,C 180,E1 -5029.332,E2 -5029.332} C_VEL
LIN {X 0,Y 516.978,Z 647.395,A -85,B 0,C 180,E1 -5030.414,E2 -5030.414} C_VEL
LIN {X 0,Y 516.758,Z 655.079,A -85,B 0,C 180,E1 -5031.396,E2 -5031.396} C_VEL
LIN {X 0,Y 516.583,Z 661.459,A -85,B 0,C 180,E1 -5032.377,E2 -5032.377} C_VEL
LIN {X 0,Y 516.461,Z 667.022,A -85,B 0,C 180,E1 -5033.407,E2 -5033.407} C_VEL
LIN {X 0,Y 516.404,Z 671.955,A -85,B 0,C 180,E1 -5034.533,E2 -5034.533} C_VEL
LIN {X 0,Y 516.364,Z 675.975,A -85,B 0,C 180,E1 -5035.707,E2 -5035.707} C_VEL
LIN {X 0,Y 516.282,Z 678.949,A -85,B 0,C 180,E1 -5036.879,E2 -5036.879} C_VEL
LIN {X 0,Y 516.192,Z 681.432,A -85,B 0,C 180,E1 -5038.44,E2 -5038.44} C_VEL
LIN {X 0,Y 516.16,Z 682.041,A -85,B 0,C 180,E1 -5039.22,E2 -5039.22} C_VEL
LIN {X 0,Y 516.16,Z 682.099,A -85,B 0,C 180,E1 -5040.78,E2 -5040.78} C_VEL
LIN {X 0,Y 516.192,Z 681.529,A -85,B 0,C 180,E1 -5041.56,E2 -5041.56} C_VEL
LIN {X 0,Y 516.283,Z 679.164,A -85,B 0,C 180,E1 -5043.121,E2 -5043.121} C_VEL
LIN {X 0,Y 516.361,Z 676.272,A -85,B 0,C 180,E1 -5044.293,E2 -5044.293} C_VEL
LIN {X 0,Y 516.404,Z 672.338,A -85,B 0,C 180,E1 -5045.467,E2 -5045.467} C_VEL
LIN {X 0,Y 516.452,Z 667.544,A -85,B 0,C 180,E1 -5046.583,E2 -5046.583} C_VEL
LIN {X 0,Y 516.576,Z 662.033,A -85,B 0,C 180,E1 -5047.623,E2 -5047.623} C_VEL
LIN {X 0,Y 516.752,Z 655.742,A -85,B 0,C 180,E1 -5048.604,E2 -5048.604} C_VEL
LIN {X 0,Y 516.95,Z 648.162,A -85,B 0,C 180,E1 -5049.587,E2 -5049.587} C_VEL
LIN {X 0,Y 517.21,Z 638.956,A -85,B 0,C 180,E1 -5050.57,E2 -5050.57} C_VEL
LIN {X 0,Y 517.512,Z 628.75,A -85,B 0,C 180,E1 -5051.456,E2 -5051.456} C_VEL
LIN {X 0,Y 517.78,Z 617.438,A -85,B 0,C 180,E1 -5052.236,E2 -5052.236} C_VEL
LIN {X 0,Y 517.991,Z 605.355,A -85,B 0,C 180,E1 -5052.887,E2 -5052.887} C_VEL
LIN {X 0,Y 518.298,Z 592.231,A -85,B 0,C 180,E1 -5053.402,E2 -5053.402} C_VEL
LIN {X 0,Y 518.487,Z 579.041,A -85,B 0,C 180,E1 -5053.747,E2 -5053.747} C_VEL
LIN {X 0,Y 518.935,Z 479.349,A -85,B 0,C 180,E1 -5055.204,E2 -5055.204} C_VEL
LIN {X 0,Y 517.489,Z 470.239,A -85,B 0,C 180,E1 -5055.4,E2 -5055.4} C_VEL
LIN {X 0,Y 517.785,Z 452.689,A -85,B 0,C 180,E1 -5058.035,E2 -5058.035} C_VEL
LIN {X 0,Y 518.146,Z 432.181,A -85,B 0,C 180,E1 -5061.066,E2 -5061.066} C_VEL
LIN {X 0,Y 518.312,Z 417.816,A -85,B 0,C 180,E1 -5063.155,E2 -5063.155} C_VEL
LIN {X 0,Y 516.873,Z 409.103,A -85,B 0,C 180,E1 -5064.478,E2 -5064.478} C_VEL
LIN {X 0,Y 516.875,Z 409.105,A -85,B 0,C 180,E1 -5067.536,E2 -5067.536} C_VEL
LIN {X 0,Y 516.869,Z 409.102,A -85,B 0,C 180,E1 -5070.205,E2 -5070.205} C_VEL
LIN {X 0,Y 516.898,Z 409.098,A -85,B 0,C 180,E1 -5072.947,E2 -5072.947} C_VEL
LIN {X 0,Y 516.87,Z 409.101,A -85,B 0,C 180,E1 -5075.781,E2 -5075.781} C_VEL
LIN {X 0,Y 516.882,Z 409.098,A -85,B 0,C 180,E1 -5078.716,E2 -5078.716} C_VEL
LIN {X 0,Y 516.914,Z 409.094,A -85,B 0,C 180,E1 -5081.775,E2 -5081.775} C_VEL
LIN {X 0,Y 516.926,Z 409.097,A -85,B 0,C 180,E1 -5085.01,E2 -5085.01} C_VEL
LIN {X 0,Y 516.916,Z 409.095,A -85,B 0,C 180,E1 -5088.399,E2 -5088.399} C_VEL
LIN {X 0,Y 516.882,Z 409.098,A -85,B 0,C 180,E1 -5091.284,E2 -5091.284} C_VEL
LIN {X 0,Y 516.87,Z 409.101,A -85,B 0,C 180,E1 -5094.219,E2 -5094.219} C_VEL
LIN {X 0,Y 516.897,Z 409.097,A -85,B 0,C 180,E1 -5097.053,E2 -5097.053} C_VEL
LIN {X 0,Y 516.869,Z 409.1,A -85,B 0,C 180,E1 -5099.795,E2 -5099.795} C_VEL
LIN {X 0,Y 516.911,Z 409.21,A -85,B 0,C 180,E1 -5102.74,E2 -5102.74} C_VEL
LIN {X 0,Y 519.121,Z 419.84,A -85,B 0,C 180,E1 -5104.327,E2 -5104.327} C_VEL
LIN {X 0,Y 518.946,Z 435.347,A -85,B 0,C 180,E1 -5106.452,E2 -5106.452} C_VEL
LIN {X 0,Y 518.301,Z 456.921,A -85,B 0,C 180,E1 -5109.356,E2 -5109.356} C_VEL
LIN {X 0,Y 517.788,Z 480.023,A -85,B 0,C 180,E1 -5112.422,E2 -5112.422} C_VEL
LIN {X 0,Y 517.408,Z 496.904,A -85,B 0,C 180,E1 -5114.638,E2 -5114.638} C_VEL
LIN {X 0,Y 518.97,Z 509.724,A -85,B 0,C 180,E1 -5114.882,E2 -5114.882} C_VEL
LIN {X 0,Y 518.538,Z 600.236,A -85,B 0,C 180,E1 -5116.154,E2 -5116.154} C_VEL
LIN {X 0,Y 518.366,Z 613.563,A -85,B 0,C 180,E1 -5116.425,E2 -5116.425} C_VEL
LIN {X 0,Y 518.096,Z 627.085,A -85,B 0,C 180,E1 -5116.867,E2 -5116.867} C_VEL
LIN {X 0,Y 517.882,Z 639.75,A -85,B 0,C 180,E1 -5117.459,E2 -5117.459} C_VEL
LIN {X 0,Y 517.6,Z 650.644,A -85,B 0,C 180,E1 -5118.122,E2 -5118.122} C_VEL
LIN {X 0,Y 517.298,Z 661.38,A -85,B 0,C 180,E1 -5118.936,E2 -5118.936} C_VEL
LIN {X 0,Y 517.04,Z 670.898,A -85,B 0,C 180,E1 -5119.822,E2 -5119.822} C_VEL
LIN {X 0,Y 516.792,Z 679.543,A -85,B 0,C 180,E1 -5120.805,E2 -5120.805} C_VEL
LIN {X 0,Y 516.605,Z 688.021,A -85,B 0,C 180,E1 -5121.984,E2 -5121.984} C_VEL
LIN {X 0,Y 516.478,Z 695.034,A -85,B 0,C 180,E1 -5123.204,E2 -5123.204} C_VEL
LIN {X 0,Y 516.402,Z 701.043,A -85,B 0,C 180,E1 -5124.533,E2 -5124.533} C_VEL
LIN {X 0,Y 516.348,Z 705.086,A -85,B 0,C 180,E1 -5125.707,E2 -5125.707} C_VEL
LIN {X 0,Y 516.313,Z 708.065,A -85,B 0,C 180,E1 -5126.879,E2 -5126.879} C_VEL
LIN {X 0,Y 516.261,Z 709.489,A -85,B 0,C 180,E1 -5127.659,E2 -5127.659} C_VEL
LIN {X 0,Y 516.178,Z 711.107,A -85,B 0,C 180,E1 -5129.22,E2 -5129.22} C_VEL
LIN {X 0,Y 516.176,Z 711.32,A -85,B 0,C 180,E1 -5130,E2 -5130} C_VEL
LIN {X 0,Y 516.179,Z 711.098,A -85,B 0,C 180,E1 -5130.78,E2 -5130.78} C_VEL
LIN {X 0,Y 516.261,Z 709.461,A -85,B 0,C 180,E1 -5132.341,E2 -5132.341} C_VEL
LIN {X 0,Y 516.313,Z 708.03,A -85,B 0,C 180,E1 -5133.121,E2 -5133.121} C_VEL
LIN {X 0,Y 516.348,Z 705.028,A -85,B 0,C 180,E1 -5134.293,E2 -5134.293} C_VEL
LIN {X 0,Y 516.402,Z 700.951,A -85,B 0,C 180,E1 -5135.467,E2 -5135.467} C_VEL
LIN {X 0,Y 516.483,Z 694.869,A -85,B 0,C 180,E1 -5136.802,E2 -5136.802} C_VEL
LIN {X 0,Y 516.605,Z 687.843,A -85,B 0,C 180,E1 -5138.016,E2 -5138.016} C_VEL
LIN {X 0,Y 516.792,Z 679.324,A -85,B 0,C 180,E1 -5139.195,E2 -5139.195} C_VEL
LIN {X 0,Y 517.04,Z 670.59,A -85,B 0,C 180,E1 -5140.178,E2 -5140.178} C_VEL
LIN {X 0,Y 517.289,Z 659.785,A -85,B 0,C 180,E1 -5141.163,E2 -5141.163} C_VEL
LIN {X 0,Y 517.564,Z 648.714,A -85,B 0,C 180,E1 -5141.974,E2 -5141.974} C_VEL
LIN {X 0,Y 517.845,Z 637.19,A -85,B 0,C 180,E1 -5142.641,E2 -5142.641} C_VEL
LIN {X 0,Y 518.088,Z 624.868,A -85,B 0,C 180,E1 -5143.183,E2 -5143.183} C_VEL
LIN {X 0,Y 518.346,Z 611.482,A -85,B 0,C 180,E1 -5143.601,E2 -5143.601} C_VEL
LIN {X 0,Y 518.543,Z 596.736,A -85,B 0,C 180,E1 -5143.87,E2 -5143.87} C_VEL
LIN {X 0,Y 518.947,Z 509.149,A -85,B 0,C 180,E1 -5145.112,E2 -5145.112} C_VEL
LIN {X 0,Y 517.383,Z 495.772,A -85,B 0,C 180,E1 -5145.374,E2 -5145.374} C_VEL
LIN {X 0,Y 517.815,Z 470.847,A -85,B 0,C 180,E1 -5148.6,E2 -5148.6} C_VEL
LIN {X 0,Y 518.259,Z 448.832,A -85,B 0,C 180,E1 -5151.478,E2 -5151.478} C_VEL
LIN {X 0,Y 518.737,Z 425.669,A -85,B 0,C 180,E1 -5154.559,E2 -5154.559} C_VEL
LIN {X 0,Y 518.766,Z 418.928,A -85,B 0,C 180,E1 -5155.476,E2 -5155.476} C_VEL
LIN {X 0,Y 516.9,Z 409.1,A -85,B 0,C 180,E1 -5156.932,E2 -5156.932} C_VEL
LIN {X 0,Y 516.869,Z 409.103,A -85,B 0,C 180,E1 -5160.205,E2 -5160.205} C_VEL
LIN {X 0,Y 516.897,Z 409.098,A -85,B 0,C 180,E1 -5162.947,E2 -5162.947} C_VEL
LIN {X 0,Y 516.869,Z 409.103,A -85,B 0,C 180,E1 -5165.781,E2 -5165.781} C_VEL
LIN {X 0,Y 516.881,Z 409.098,A -85,B 0,C 180,E1 -5168.716,E2 -5168.716} C_VEL
LIN {X 0,Y 516.909,Z 409.095,A -85,B 0,C 180,E1 -5171.776,E2 -5171.776} C_VEL
LIN {X 0,Y 516.926,Z 409.097,A -85,B 0,C 180,E1 -5175.01,E2 -5175.01} C_VEL
LIN {X 0,Y 516.916,Z 409.092,A -85,B 0,C 180,E1 -5178.399,E2 -5178.399} C_VEL
LIN {X 0,Y 516.884,Z 409.102,A -85,B 0,C 180,E1 -5181.284,E2 -5181.284} C_VEL
LIN {X 0,Y 516.875,Z 409.097,A -85,B 0,C 180,E1 -5184.22,E2 -5184.22} C_VEL
LIN {X 0,Y 516.898,Z 409.1,A -85,B 0,C 180,E1 -5187.053,E2 -5187.053} C_VEL
LIN {X 0,Y 516.895,Z 409.095,A -85,B 0,C 180,E1 -5189.796,E2 -5189.796} C_VEL
LIN {X 0,Y 516.927,Z 409.096,A -85,B 0,C 180,E1 -5192.467,E2 -5192.467} C_VEL
LIN {X 0,Y 516.876,Z 409.104,A -85,B 0,C 180,E1 -5195.07,E2 -5195.07} C_VEL
LIN {X 0,Y 516.872,Z 409.1,A -85,B 0,C 180,E1 -5197.622,E2 -5197.622} C_VEL
LIN {X 0,Y 516.932,Z 409.094,A -85,B 0,C 180,E1 -5200.13,E2 -5200.13} C_VEL
LIN {X 0,Y 516.897,Z 409.102,A -85,B 0,C 180,E1 -5202.595,E2 -5202.595} C_VEL
LIN {X 0,Y 516.928,Z 409.098,A -85,B 0,C 180,E1 -5204.773,E2 -5204.773} C_VEL
LIN {X 0,Y 519.151,Z 416.421,A -85,B 0,C 180,E1 -5204.958,E2 -5204.958} C_VEL
LIN {X 0,Y 518.541,Z 512.329,A -85,B 0,C 180,E1 -5206.379,E2 -5206.379} C_VEL
LIN {X 0,Y 518.371,Z 525.83,A -85,B 0,C 180,E1 -5206.749,E2 -5206.749} C_VEL
LIN {X 0,Y 518.139,Z 538.505,A -85,B 0,C 180,E1 -5207.267,E2 -5207.267} C_VEL
LIN {X 0,Y 517.882,Z 551.128,A -85,B 0,C 180,E1 -5207.97,E2 -5207.97} C_VEL
LIN {X 0,Y 517.61,Z 561.955,A -85,B 0,C 180,E1 -5208.745,E2 -5208.745} C_VEL
LIN {X 0,Y 517.361,Z 571.836,A -85,B 0,C 180,E1 -5209.631,E2 -5209.631} C_VEL
LIN {X 0,Y 517.119,Z 580.788,A -85,B 0,C 180,E1 -5210.614,E2 -5210.614} C_VEL
LIN {X 0,Y 516.841,Z 589.492,A -85,B 0,C 180,E1 -5211.791,E2 -5211.791} C_VEL
LIN {X 0,Y 516.664,Z 596.387,A -85,B 0,C 180,E1 -5212.968,E2 -5212.968} C_VEL
LIN {X 0,Y 516.583,Z 601.899,A -85,B 0,C 180,E1 -5214.144,E2 -5214.144} C_VEL
LIN {X 0,Y 516.408,Z 606.239,A -85,B 0,C 180,E1 -5215.316,E2 -5215.316} C_VEL
LIN {X 0,Y 516.437,Z 608.497,A -85,B 0,C 180,E1 -5216.098,E2 -5216.098} C_VEL
LIN {X 0,Y 516.37,Z 610.364,A -85,B 0,C 180,E1 -5216.879,E2 -5216.879} C_VEL
LIN {X 0,Y 516.289,Z 611.776,A -85,B 0,C 180,E1 -5217.66,E2 -5217.66} C_VEL
LIN {X 0,Y 516.218,Z 613.365,A -85,B 0,C 180,E1 -5219.22,E2 -5219.22} C_VEL
LIN {X 0,Y 516.213,Z 613.587,A -85,B 0,C 180,E1 -5220,E2 -5220} C_VEL
LIN {X 0,Y 516.23,Z 612.778,A -85,B 0,C 180,E1 -5221.56,E2 -5221.56} C_VEL
LIN {X 0,Y 516.281,Z 611.829,A -85,B 0,C 180,E1 -5222.341,E2 -5222.341} C_VEL
LIN {X 0,Y 516.365,Z 610.432,A -85,B 0,C 180,E1 -5223.121,E2 -5223.121} C_VEL
LIN {X 0,Y 516.439,Z 607.565,A -85,B 0,C 180,E1 -5224.293,E2 -5224.293} C_VEL
LIN {X 0,Y 516.43,Z 603.678,A -85,B 0,C 180,E1 -5225.466,E2 -5225.466} C_VEL
LIN {X 0,Y 516.573,Z 598.335,A -85,B 0,C 180,E1 -5226.699,E2 -5226.699} C_VEL
LIN {X 0,Y 516.743,Z 592.241,A -85,B 0,C 180,E1 -5227.817,E2 -5227.817} C_VEL
LIN {X 0,Y 516.961,Z 584.315,A -85,B 0,C 180,E1 -5228.995,E2 -5228.995} C_VEL
LIN {X 0,Y 517.186,Z 576.185,A -85,B 0,C 180,E1 -5229.977,E2 -5229.977} C_VEL
LIN {X 0,Y 517.439,Z 566.219,A -85,B 0,C 180,E1 -5230.962,E2 -5230.962} C_VEL
LIN {X 0,Y 517.728,Z 556.322,A -85,B 0,C 180,E1 -5231.749,E2 -5231.749} C_VEL
LIN {X 0,Y 517.987,Z 544.892,A -85,B 0,C 180,E1 -5232.48,E2 -5232.48} C_VEL
LIN {X 0,Y 518.219,Z 532.671,A -85,B 0,C 180,E1 -5233.08,E2 -5233.08} C_VEL
LIN {X 0,Y 518.45,Z 520.079,A -85,B 0,C 180,E1 -5233.523,E2 -5233.523} C_VEL
LIN {X 0,Y 518.583,Z 507.1,A -85,B 0,C 180,E1 -5233.819,E2 -5233.819} C_VEL
LIN {X 0,Y 518.987,Z 415.569,A -85,B 0,C 180,E1 -5235.143,E2 -5235.143} C_VEL
LIN {X 0,Y 516.905,Z 409.1,A -85,B 0,C 180,E1 -5235.317,E2 -5235.317} C_VEL
LIN {X 0,Y 516.881,Z 409.099,A -85,B 0,C 180,E1 -5238.224,E2 -5238.224} C_VEL
LIN {X 0,Y 516.908,Z 409.095,A -85,B 0,C 180,E1 -5240.702,E2 -5240.702} C_VEL
LIN {X 0,Y 516.889,Z 409.095,A -85,B 0,C 180,E1 -5244.073,E2 -5244.073} C_VEL
LIN {X 0,Y 516.907,Z 409.093,A -85,B 0,C 180,E1 -5246.659,E2 -5246.659} C_VEL
LIN {X 0,Y 516.913,Z 409.096,A -85,B 0,C 180,E1 -5249.524,E2 -5249.524} C_VEL
LIN {X 0,Y 516.899,Z 409.092,A -85,B 0,C 180,E1 -5252.543,E2 -5252.543} C_VEL
LIN {X 0,Y 516.869,Z 409.102,A -85,B 0,C 180,E1 -5255.33,E2 -5255.33} C_VEL
LIN {X 0,Y 516.879,Z 409.099,A -85,B 0,C 180,E1 -5256.643,E2 -5256.643} C_VEL
LIN {X 0,Y 516.245,Z 409.184,A -85,B 0,C 180,E1 -5257.293,E2 -5257.293} C_VEL
LIN {X 0,Y 513.378,Z 409.536,A -85,B 0,C 180,E1 -5258.347,E2 -5258.347} C_VEL
LIN {X 0,Y 510.939,Z 409.837,A -85,B 0,C 180,E1 -5259.197,E2 -5259.197} C_VEL
LIN {X 0,Y 509.902,Z 409.961,A -85,B 0,C 180,E1 -5259.853,E2 -5259.853} C_VEL
LIN {X 0,Y 509.825,Z 409.97,A -85,B 0,C 180,E1 -5260.075,E2 -5260.075} C_VEL
LIN {X 0,Y 509.836,Z 409.976,A -85,B 0,C 180,E1 -5262.49,E2 -5262.49} C_VEL
LIN {X 0,Y 509.86,Z 409.967,A -85,B 0,C 180,E1 -5265.332,E2 -5265.332} C_VEL
LIN {X 0,Y 509.858,Z 409.978,A -85,B 0,C 180,E1 -5268.575,E2 -5268.575} C_VEL
LIN {X 0,Y 509.852,Z 409.972,A -85,B 0,C 180,E1 -5271.787,E2 -5271.787} C_VEL
LIN {X 0,Y 509.83,Z 409.982,A -85,B 0,C 180,E1 -5274.622,E2 -5274.622} C_VEL
LIN {X 0,Y 509.864,Z 409.971,A -85,B 0,C 180,E1 -5277.481,E2 -5277.481} C_VEL
LIN {X 0,Y 509.855,Z 409.979,A -85,B 0,C 180,E1 -5280.275,E2 -5280.275} C_VEL
LIN {X 0,Y 509.824,Z 409.981,A -85,B 0,C 180,E1 -5282.941,E2 -5282.941} C_VEL
LIN {X 0,Y 509.841,Z 410.116,A -85,B 0,C 180,E1 -5285.157,E2 -5285.157} C_VEL
LIN {X 0,Y 511.464,Z 418.443,A -85,B 0,C 180,E1 -5286.516,E2 -5286.516} C_VEL
LIN {X 0,Y 511.472,Z 426.562,A -85,B 0,C 180,E1 -5287.798,E2 -5287.798} C_VEL
LIN {X 0,Y 510.985,Z 445.41,A -85,B 0,C 180,E1 -5290.726,E2 -5290.726} C_VEL
LIN {X 0,Y 510.58,Z 465.805,A -85,B 0,C 180,E1 -5293.815,E2 -5293.815} C_VEL
LIN {X 0,Y 510.515,Z 470.238,A -85,B 0,C 180,E1 -5294.455,E2 -5294.455} C_VEL
LIN {X 0,Y 512.215,Z 481.076,A -85,B 0,C 180,E1 -5294.678,E2 -5294.678} C_VEL
LIN {X 0,Y 511.754,Z 578.463,A -85,B 0,C 180,E1 -5296.069,E2 -5296.069} C_VEL
LIN {X 0,Y 511.503,Z 592.006,A -85,B 0,C 180,E1 -5296.416,E2 -5296.416} C_VEL
LIN {X 0,Y 511.236,Z 605.149,A -85,B 0,C 180,E1 -5296.94,E2 -5296.94} C_VEL
LIN {X 0,Y 510.926,Z 617.202,A -85,B 0,C 180,E1 -5297.591,E2 -5297.591} C_VEL
LIN {X 0,Y 510.692,Z 628.56,A -85,B 0,C 180,E1 -5298.389,E2 -5298.389} C_VEL
LIN {X 0,Y 510.249,Z 639.811,A -85,B 0,C 180,E1 -5299.384,E2 -5299.384} C_VEL
LIN {X 0,Y 509.97,Z 648.041,A -85,B 0,C 180,E1 -5300.281,E2 -5300.281} C_VEL
LIN {X 0,Y 509.727,Z 656.975,A -85,B 0,C 180,E1 -5301.476,E2 -5301.476} C_VEL
LIN {X 0,Y 509.501,Z 664.148,A -85,B 0,C 180,E1 -5302.669,E2 -5302.669} C_VEL
LIN {X 0,Y 509.397,Z 669.018,A -85,B 0,C 180,E1 -5303.663,E2 -5303.663} C_VEL
LIN {X 0,Y 509.248,Z 673.732,A -85,B 0,C 180,E1 -5304.853,E2 -5304.853} C_VEL
LIN {X 0,Y 509.303,Z 677.338,A -85,B 0,C 180,E1 -5306.044,E2 -5306.044} C_VEL
LIN {X 0,Y 509.201,Z 679.198,A -85,B 0,C 180,E1 -5306.835,E2 -5306.835} C_VEL
LIN {X 0,Y 509.19,Z 680.622,A -85,B 0,C 180,E1 -5307.627,E2 -5307.627} C_VEL
LIN {X 0,Y 509.074,Z 682.237,A -85,B 0,C 180,E1 -5309.209,E2 -5309.209} C_VEL
LIN {X 0,Y 509.066,Z 682.476,A -85,B 0,C 180,E1 -5310,E2 -5310} C_VEL
LIN {X 0,Y 509.073,Z 682.291,A -85,B 0,C 180,E1 -5310.791,E2 -5310.791} C_VEL
LIN {X 0,Y 509.19,Z 680.746,A -85,B 0,C 180,E1 -5312.373,E2 -5312.373} C_VEL
LIN {X 0,Y 509.202,Z 679.39,A -85,B 0,C 180,E1 -5313.165,E2 -5313.165} C_VEL
LIN {X 0,Y 509.283,Z 676.533,A -85,B 0,C 180,E1 -5314.353,E2 -5314.353} C_VEL
LIN {X 0,Y 509.345,Z 672.653,A -85,B 0,C 180,E1 -5315.543,E2 -5315.543} C_VEL
LIN {X 0,Y 509.431,Z 666.918,A -85,B 0,C 180,E1 -5316.878,E2 -5316.878} C_VEL
LIN {X 0,Y 509.629,Z 660.092,A -85,B 0,C 180,E1 -5318.126,E2 -5318.126} C_VEL
LIN {X 0,Y 509.844,Z 651.948,A -85,B 0,C 180,E1 -5319.321,E2 -5319.321} C_VEL
LIN {X 0,Y 510.097,Z 643.559,A -85,B 0,C 180,E1 -5320.318,E2 -5320.318} C_VEL
LIN {X 0,Y 510.511,Z 633.261,A -85,B 0,C 180,E1 -5321.313,E2 -5321.313} C_VEL
LIN {X 0,Y 510.829,Z 622.076,A -85,B 0,C 180,E1 -5322.18,E2 -5322.18} C_VEL
LIN {X 0,Y 511.153,Z 609.957,A -85,B 0,C 180,E1 -5322.91,E2 -5322.91} C_VEL
LIN {X 0,Y 511.432,Z 597.975,A -85,B 0,C 180,E1 -5323.459,E2 -5323.459} C_VEL
LIN {X 0,Y 511.662,Z 584.657,A -85,B 0,C 180,E1 -5323.883,E2 -5323.883} C_VEL
LIN {X 0,Y 511.829,Z 571.847,A -85,B 0,C 180,E1 -5324.132,E2 -5324.132} C_VEL
LIN {X 0,Y 512.183,Z 480.278,A -85,B 0,C 180,E1 -5325.425,E2 -5325.425} C_VEL
LIN {X 0,Y 510.536,Z 470.21,A -85,B 0,C 180,E1 -5325.624,E2 -5325.624} C_VEL
LIN {X 0,Y 510.905,Z 450.079,A -85,B 0,C 180,E1 -5328.653,E2 -5328.653} C_VEL
LIN {X 0,Y 511.298,Z 432.549,A -85,B 0,C 180,E1 -5331.362,E2 -5331.362} C_VEL
LIN {X 0,Y 511.529,Z 418.992,A -85,B 0,C 180,E1 -5333.481,E2 -5333.481} C_VEL
LIN {X 0,Y 509.817,Z 409.982,A -85,B 0,C 180,E1 -5334.98,E2 -5334.98} C_VEL
LIN {X 0,Y 509.837,Z 409.98,A -85,B 0,C 180,E1 -5337.949,E2 -5337.949} C_VEL
LIN {X 0,Y 509.837,Z 409.975,A -85,B 0,C 180,E1 -5340.667,E2 -5340.667} C_VEL
LIN {X 0,Y 509.862,Z 409.979,A -85,B 0,C 180,E1 -5343.461,E2 -5343.461} C_VEL
LIN {X 0,Y 509.812,Z 409.978,A -85,B 0,C 180,E1 -5346.354,E2 -5346.354} C_VEL
LIN {X 0,Y 509.848,Z 409.977,A -85,B 0,C 180,E1 -5349.352,E2 -5349.352} C_VEL
LIN {X 0,Y 509.836,Z 409.975,A -85,B 0,C 180,E1 -5352.49,E2 -5352.49} C_VEL
LIN {X 0,Y 509.86,Z 409.976,A -85,B 0,C 180,E1 -5355.332,E2 -5355.332} C_VEL
LIN {X 0,Y 509.858,Z 409.972,A -85,B 0,C 180,E1 -5358.574,E2 -5358.574} C_VEL
LIN {X 0,Y 509.854,Z 409.971,A -85,B 0,C 180,E1 -5361.787,E2 -5361.787} C_VEL
LIN {X 0,Y 509.83,Z 409.976,A -85,B 0,C 180,E1 -5364.622,E2 -5364.622} C_VEL
LIN {X 0,Y 509.864,Z 409.97,A -85,B 0,C 180,E1 -5367.481,E2 -5367.481} C_VEL
LIN {X 0,Y 509.856,Z 409.978,A -85,B 0,C 180,E1 -5370.275,E2 -5370.275} C_VEL
LIN {X 0,Y 509.827,Z 409.978,A -85,B 0,C 180,E1 -5372.941,E2 -5372.941} C_VEL
LIN {X 0,Y 509.847,Z 410.149,A -85,B 0,C 180,E1 -5375.157,E2 -5375.157} C_VEL
LIN {X 0,Y 511.477,Z 418.444,A -85,B 0,C 180,E1 -5376.517,E2 -5376.517} C_VEL
LIN {X 0,Y 511.426,Z 428.057,A -85,B 0,C 180,E1 -5378.008,E2 -5378.008} C_VEL
LIN {X 0,Y 511.015,Z 447.089,A -85,B 0,C 180,E1 -5380.935,E2 -5380.935} C_VEL
LIN {X 0,Y 510.567,Z 467.323,A -85,B 0,C 180,E1 -5384.02,E2 -5384.02} C_VEL
LIN {X 0,Y 510.494,Z 470.316,A -85,B 0,C 180,E1 -5384.481,E2 -5384.481} C_VEL
LIN {X 0,Y 512.158,Z 480.708,A -85,B 0,C 180,E1 -5384.7,E2 -5384.7} C_VEL
LIN {X 0,Y 511.595,Z 579.635,A -85,B 0,C 180,E1 -5386.165,E2 -5386.165} C_VEL
LIN {X 0,Y 511.37,Z 593.254,A -85,B 0,C 180,E1 -5386.539,E2 -5386.539} C_VEL
LIN {X 0,Y 511.099,Z 605.536,A -85,B 0,C 180,E1 -5387.038,E2 -5387.038} C_VEL
LIN {X 0,Y 510.831,Z 617.487,A -85,B 0,C 180,E1 -5387.691,E2 -5387.691} C_VEL
LIN {X 0,Y 510.528,Z 628.843,A -85,B 0,C 180,E1 -5388.486,E2 -5388.486} C_VEL
LIN {X 0,Y 510.217,Z 639.044,A -85,B 0,C 180,E1 -5389.383,E2 -5389.383} C_VEL
LIN {X 0,Y 509.977,Z 647.421,A -85,B 0,C 180,E1 -5390.281,E2 -5390.281} C_VEL
LIN {X 0,Y 509.732,Z 655.147,A -85,B 0,C 180,E1 -5391.277,E2 -5391.277} C_VEL
LIN {X 0,Y 509.497,Z 662.729,A -85,B 0,C 180,E1 -5392.47,E2 -5392.47} C_VEL
LIN {X 0,Y 509.368,Z 668.818,A -85,B 0,C 180,E1 -5393.663,E2 -5393.663} C_VEL
LIN {X 0,Y 509.251,Z 673.6,A -85,B 0,C 180,E1 -5394.853,E2 -5394.853} C_VEL
LIN {X 0,Y 509.304,Z 677.262,A -85,B 0,C 180,E1 -5396.044,E2 -5396.044} C_VEL
LIN {X 0,Y 509.202,Z 679.12,A -85,B 0,C 180,E1 -5396.835,E2 -5396.835} C_VEL
LIN {X 0,Y 509.19,Z 680.555,A -85,B 0,C 180,E1 -5397.627,E2 -5397.627} C_VEL
LIN {X 0,Y 509.112,Z 681.611,A -85,B 0,C 180,E1 -5398.418,E2 -5398.418} C_VEL
LIN {X 0,Y 509.074,Z 682.229,A -85,B 0,C 180,E1 -5399.209,E2 -5399.209} C_VEL
LIN {X 0,Y 509.073,Z 682.289,A -85,B 0,C 180,E1 -5400.791,E2 -5400.791} C_VEL
LIN {X 0,Y 509.113,Z 681.713,A -85,B 0,C 180,E1 -5401.582,E2 -5401.582} C_VEL
LIN {X 0,Y 509.202,Z 679.343,A -85,B 0,C 180,E1 -5403.165,E2 -5403.165} C_VEL
LIN {X 0,Y 509.282,Z 676.439,A -85,B 0,C 180,E1 -5404.353,E2 -5404.353} C_VEL
LIN {X 0,Y 509.346,Z 672.489,A -85,B 0,C 180,E1 -5405.543,E2 -5405.543} C_VEL
LIN {X 0,Y 509.417,Z 666.753,A -85,B 0,C 180,E1 -5406.864,E2 -5406.864} C_VEL
LIN {X 0,Y 509.609,Z 659.782,A -85,B 0,C 180,E1 -5408.126,E2 -5408.126} C_VEL
LIN {X 0,Y 509.808,Z 651.424,A -85,B 0,C 180,E1 -5409.322,E2 -5409.322} C_VEL
LIN {X 0,Y 510.047,Z 642.868,A -85,B 0,C 180,E1 -5410.319,E2 -5410.319} C_VEL
LIN {X 0,Y 510.412,Z 633.466,A -85,B 0,C 180,E1 -5411.215,E2 -5411.215} C_VEL
LIN {X 0,Y 510.678,Z 622.958,A -85,B 0,C 180,E1 -5412.03,E2 -5412.03} C_VEL
LIN {X 0,Y 510.959,Z 611.909,A -85,B 0,C 180,E1 -5412.713,E2 -5412.713} C_VEL
LIN {X 0,Y 511.177,Z 600.464,A -85,B 0,C 180,E1 -5413.264,E2 -5413.264} C_VEL
LIN {X 0,Y 511.407,Z 587.421,A -85,B 0,C 180,E1 -5413.713,E2 -5413.713} C_VEL
LIN {X 0,Y 511.631,Z 575.169,A -85,B 0,C 180,E1 -5413.986,E2 -5413.986} C_VEL
LIN {X 0,Y 512.109,Z 480.32,A -85,B 0,C 180,E1 -5415.395,E2 -5415.395} C_VEL
LIN {X 0,Y 510.539,Z 470.556,A -85,B 0,C 180,E1 -5415.598,E2 -5415.598} C_VEL
LIN {X 0,Y 510.93,Z 450.187,A -85,B 0,C 180,E1 -5418.652,E2 -5418.652} C_VEL
LIN {X 0,Y 511.271,Z 430.483,A -85,B 0,C 180,E1 -5421.574,E2 -5421.574} C_VEL
LIN {X 0,Y 511.373,Z 418.633,A -85,B 0,C 180,E1 -5423.325,E2 -5423.325} C_VEL
LIN {X 0,Y 509.83,Z 409.98,A -85,B 0,C 180,E1 -5424.652,E2 -5424.652} C_VEL
LIN {X 0,Y 509.823,Z 409.98,A -85,B 0,C 180,E1 -5427.059,E2 -5427.059} C_VEL
LIN {X 0,Y 509.854,Z 409.98,A -85,B 0,C 180,E1 -5429.751,E2 -5429.751} C_VEL
LIN {X 0,Y 509.876,Z 409.971,A -85,B 0,C 180,E1 -5432.774,E2 -5432.774} C_VEL
LIN {X 0,Y 509.826,Z 409.981,A -85,B 0,C 180,E1 -5435.578,E2 -5435.578} C_VEL
LIN {X 0,Y 509.851,Z 409.972,A -85,B 0,C 180,E1 -5438.338,E2 -5438.338} C_VEL
LIN {X 0,Y 509.858,Z 409.976,A -85,B 0,C 180,E1 -5441.425,E2 -5441.425} C_VEL
LIN {X 0,Y 509.86,Z 409.976,A -85,B 0,C 180,E1 -5444.668,E2 -5444.668} C_VEL
LIN {X 0,Y 509.858,Z 409.972,A -85,B 0,C 180,E1 -5448.103,E2 -5448.103} C_VEL
LIN {X 0,Y 509.848,Z 409.978,A -85,B 0,C 180,E1 -5450.647,E2 -5450.647} C_VEL
LIN {X 0,Y 509.811,Z 409.977,A -85,B 0,C 180,E1 -5453.646,E2 -5453.646} C_VEL
LIN {X 0,Y 509.861,Z 409.977,A -85,B 0,C 180,E1 -5456.539,E2 -5456.539} C_VEL
LIN {X 0,Y 509.836,Z 409.976,A -85,B 0,C 180,E1 -5459.333,E2 -5459.333} C_VEL
LIN {X 0,Y 509.871,Z 410.026,A -85,B 0,C 180,E1 -5462.527,E2 -5462.527} C_VEL
LIN {X 0,Y 512.326,Z 422.445,A -85,B 0,C 180,E1 -5464.398,E2 -5464.398} C_VEL
LIN {X 0,Y 511.787,Z 440.807,A -85,B 0,C 180,E1 -5466.936,E2 -5466.936} C_VEL
LIN {X 0,Y 511.32,Z 457.988,A -85,B 0,C 180,E1 -5469.279,E2 -5469.279} C_VEL
LIN {X 0,Y 510.761,Z 481.012,A -85,B 0,C 180,E1 -5472.379,E2 -5472.379} C_VEL
LIN {X 0,Y 510.382,Z 496.24,A -85,B 0,C 180,E1 -5474.409,E2 -5474.409} C_VEL
LIN {X 0,Y 512.087,Z 510.358,A -85,B 0,C 180,E1 -5474.693,E2 -5474.693} C_VEL
LIN {X 0,Y 511.623,Z 600.116,A -85,B 0,C 180,E1 -5475.989,E2 -5475.989} C_VEL
LIN {X 0,Y 511.404,Z 614.12,A -85,B 0,C 180,E1 -5476.287,E2 -5476.287} C_VEL
LIN {X 0,Y 511.122,Z 627.245,A -85,B 0,C 180,E1 -5476.735,E2 -5476.735} C_VEL
LIN {X 0,Y 510.864,Z 638.782,A -85,B 0,C 180,E1 -5477.284,E2 -5477.284} C_VEL
LIN {X 0,Y 510.567,Z 650.341,A -85,B 0,C 180,E1 -5477.998,E2 -5477.998} C_VEL
LIN {X 0,Y 510.244,Z 661.728,A -85,B 0,C 180,E1 -5478.882,E2 -5478.882} C_VEL
LIN {X 0,Y 509.933,Z 671.928,A -85,B 0,C 180,E1 -5479.879,E2 -5479.879} C_VEL
LIN {X 0,Y 509.683,Z 680.339,A -85,B 0,C 180,E1 -5480.876,E2 -5480.876} C_VEL
LIN {X 0,Y 509.513,Z 688.542,A -85,B 0,C 180,E1 -5482.072,E2 -5482.072} C_VEL
LIN {X 0,Y 509.383,Z 695.092,A -85,B 0,C 180,E1 -5483.265,E2 -5483.265} C_VEL
LIN {X 0,Y 509.338,Z 700.347,A -85,B 0,C 180,E1 -5484.457,E2 -5484.457} C_VEL
LIN {X 0,Y 509.273,Z 704.415,A -85,B 0,C 180,E1 -5485.647,E2 -5485.647} C_VEL
LIN {X 0,Y 509.259,Z 707.399,A -85,B 0,C 180,E1 -5486.836,E2 -5486.836} C_VEL
LIN {X 0,Y 509.191,Z 708.836,A -85,B 0,C 180,E1 -5487.627,E2 -5487.627} C_VEL
LIN {X 0,Y 509.109,Z 710.434,A -85,B 0,C 180,E1 -5489.209,E2 -5489.209} C_VEL
LIN {X 0,Y 509.108,Z 710.655,A -85,B 0,C 180,E1 -5490,E2 -5490} C_VEL
LIN {X 0,Y 509.11,Z 710.429,A -85,B 0,C 180,E1 -5490.791,E2 -5490.791} C_VEL
LIN {X 0,Y 509.134,Z 709.796,A -85,B 0,C 180,E1 -5491.582,E2 -5491.582} C_VEL
LIN {X 0,Y 509.259,Z 707.321,A -85,B 0,C 180,E1 -5493.164,E2 -5493.164} C_VEL
LIN {X 0,Y 509.274,Z 704.285,A -85,B 0,C 180,E1 -5494.353,E2 -5494.353} C_VEL
LIN {X 0,Y 509.338,Z 700.17,A -85,B 0,C 180,E1 -5495.543,E2 -5495.543} C_VEL
LIN {X 0,Y 509.404,Z 694.315,A -85,B 0,C 180,E1 -5496.844,E2 -5496.844} C_VEL
LIN {X 0,Y 509.513,Z 688.23,A -85,B 0,C 180,E1 -5497.928,E2 -5497.928} C_VEL
LIN {X 0,Y 509.683,Z 679.99,A -85,B 0,C 180,E1 -5499.124,E2 -5499.124} C_VEL
LIN {X 0,Y 509.992,Z 669.629,A -85,B 0,C 180,E1 -5500.32,E2 -5500.32} C_VEL
LIN {X 0,Y 510.259,Z 658.749,A -85,B 0,C 180,E1 -5501.319,E2 -5501.319} C_VEL
LIN {X 0,Y 510.508,Z 647.514,A -85,B 0,C 180,E1 -5502.142,E2 -5502.142} C_VEL
LIN {X 0,Y 510.85,Z 635.931,A -85,B 0,C 180,E1 -5502.817,E2 -5502.817} C_VEL
LIN {X 0,Y 511.138,Z 623.469,A -85,B 0,C 180,E1 -5503.366,E2 -5503.366} C_VEL
LIN {X 0,Y 511.428,Z 609.711,A -85,B 0,C 180,E1 -5503.788,E2 -5503.788} C_VEL
LIN {X 0,Y 511.59,Z 594.285,A -85,B 0,C 180,E1 -5504.063,E2 -5504.063} C_VEL
LIN {X 0,Y 511.999,Z 508.888,A -85,B 0,C 180,E1 -5505.312,E2 -5505.312} C_VEL
LIN {X 0,Y 510.32,Z 494.959,A -85,B 0,C 180,E1 -5505.583,E2 -5505.583} C_VEL
LIN {X 0,Y 510.767,Z 471.542,A -85,B 0,C 180,E1 -5508.658,E2 -5508.658} C_VEL
LIN {X 0,Y 511.263,Z 449.58,A -85,B 0,C 180,E1 -5511.575,E2 -5511.575} C_VEL
LIN {X 0,Y 511.794,Z 426.525,A -85,B 0,C 180,E1 -5514.698,E2 -5514.698} C_VEL
LIN {X 0,Y 511.788,Z 419.801,A -85,B 0,C 180,E1 -5515.631,E2 -5515.631} C_VEL
LIN {X 0,Y 509.847,Z 409.979,A -85,B 0,C 180,E1 -5517.113,E2 -5517.113} C_VEL
LIN {X 0,Y 509.854,Z 409.981,A -85,B 0,C 180,E1 -5519.751,E2 -5519.751} C_VEL
LIN {X 0,Y 509.875,Z 409.972,A -85,B 0,C 180,E1 -5522.774,E2 -5522.774} C_VEL
LIN {X 0,Y 509.824,Z 409.983,A -85,B 0,C 180,E1 -5525.578,E2 -5525.578} C_VEL
LIN {X 0,Y 509.851,Z 409.973,A -85,B 0,C 180,E1 -5528.338,E2 -5528.338} C_VEL
LIN {X 0,Y 509.855,Z 409.979,A -85,B 0,C 180,E1 -5531.426,E2 -5531.426} C_VEL
LIN {X 0,Y 509.859,Z 409.973,A -85,B 0,C 180,E1 -5534.668,E2 -5534.668} C_VEL
LIN {X 0,Y 509.858,Z 409.971,A -85,B 0,C 180,E1 -5538.103,E2 -5538.103} C_VEL
LIN {X 0,Y 509.849,Z 409.975,A -85,B 0,C 180,E1 -5540.648,E2 -5540.648} C_VEL
LIN {X 0,Y 509.828,Z 409.976,A -85,B 0,C 180,E1 -5543.647,E2 -5543.647} C_VEL
LIN {X 0,Y 509.863,Z 409.973,A -85,B 0,C 180,E1 -5546.539,E2 -5546.539} C_VEL
LIN {X 0,Y 509.848,Z 409.976,A -85,B 0,C 180,E1 -5549.334,E2 -5549.334} C_VEL
LIN {X 0,Y 509.888,Z 409.969,A -85,B 0,C 180,E1 -5552.054,E2 -5552.054} C_VEL
LIN {X 0,Y 509.841,Z 409.982,A -85,B 0,C 180,E1 -5554.702,E2 -5554.702} C_VEL
LIN {X 0,Y 509.83,Z 409.978,A -85,B 0,C 180,E1 -5557.458,E2 -5557.458} C_VEL
LIN {X 0,Y 509.919,Z 409.966,A -85,B 0,C 180,E1 -5559.845,E2 -5559.845} C_VEL
LIN {X 0,Y 509.861,Z 409.975,A -85,B 0,C 180,E1 -5563.174,E2 -5563.174} C_VEL
LIN {X 0,Y 509.87,Z 410.11,A -85,B 0,C 180,E1 -5564.571,E2 -5564.571} C_VEL
LIN {X 0,Y 512.32,Z 417.602,A -85,B 0,C 180,E1 -5564.766,E2 -5564.766} C_VEL
LIN {X 0,Y 511.639,Z 513.066,A -85,B 0,C 180,E1 -5566.217,E2 -5566.217} C_VEL
LIN {X 0,Y 511.457,Z 526.553,A -85,B 0,C 180,E1 -5566.592,E2 -5566.592} C_VEL
LIN {X 0,Y 511.247,Z 538.745,A -85,B 0,C 180,E1 -5567.092,E2 -5567.092} C_VEL
LIN {X 0,Y 510.985,Z 550.81,A -85,B 0,C 180,E1 -5567.763,E2 -5567.763} C_VEL
LIN {X 0,Y 510.676,Z 562.394,A -85,B 0,C 180,E1 -5568.59,E2 -5568.59} C_VEL
LIN {X 0,Y 510.411,Z 572.36,A -85,B 0,C 180,E1 -5569.488,E2 -5569.488} C_VEL
LIN {X 0,Y 510.142,Z 581.346,A -85,B 0,C 180,E1 -5570.484,E2 -5570.484} C_VEL
LIN {X 0,Y 509.853,Z 590.082,A -85,B 0,C 180,E1 -5571.678,E2 -5571.678} C_VEL
LIN {X 0,Y 509.653,Z 597.034,A -85,B 0,C 180,E1 -5572.871,E2 -5572.871} C_VEL
LIN {X 0,Y 509.561,Z 602.562,A -85,B 0,C 180,E1 -5574.063,E2 -5574.063} C_VEL
LIN {X 0,Y 509.366,Z 606.907,A -85,B 0,C 180,E1 -5575.251,E2 -5575.251} C_VEL
LIN {X 0,Y 509.399,Z 609.174,A -85,B 0,C 180,E1 -5576.044,E2 -5576.044} C_VEL
LIN {X 0,Y 509.313,Z 611.041,A -85,B 0,C 180,E1 -5576.836,E2 -5576.836} C_VEL
LIN {X 0,Y 509.228,Z 612.455,A -85,B 0,C 180,E1 -5577.627,E2 -5577.627} C_VEL
LIN {X 0,Y 509.151,Z 614.042,A -85,B 0,C 180,E1 -5579.209,E2 -5579.209} C_VEL
LIN {X 0,Y 509.146,Z 614.261,A -85,B 0,C 180,E1 -5580,E2 -5580} C_VEL
LIN {X 0,Y 509.15,Z 614.062,A -85,B 0,C 180,E1 -5580.791,E2 -5580.791} C_VEL
LIN {X 0,Y 509.216,Z 612.474,A -85,B 0,C 180,E1 -5582.373,E2 -5582.373} C_VEL
LIN {X 0,Y 509.309,Z 611.078,A -85,B 0,C 180,E1 -5583.164,E2 -5583.164} C_VEL
LIN {X 0,Y 509.398,Z 608.183,A -85,B 0,C 180,E1 -5584.352,E2 -5584.352} C_VEL
LIN {X 0,Y 509.386,Z 604.269,A -85,B 0,C 180,E1 -5585.542,E2 -5585.542} C_VEL
LIN {X 0,Y 509.536,Z 599.177,A -85,B 0,C 180,E1 -5586.736,E2 -5586.736} C_VEL
LIN {X 0,Y 509.728,Z 592.782,A -85,B 0,C 180,E1 -5587.925,E2 -5587.925} C_VEL
LIN {X 0,Y 509.956,Z 584.795,A -85,B 0,C 180,E1 -5589.119,E2 -5589.119} C_VEL
LIN {X 0,Y 510.215,Z 576.618,A -85,B 0,C 180,E1 -5590.115,E2 -5590.115} C_VEL
LIN {X 0,Y 510.48,Z 566.606,A -85,B 0,C 180,E1 -5591.113,E2 -5591.113} C_VEL
LIN {X 0,Y 510.841,Z 555.542,A -85,B 0,C 180,E1 -5591.989,E2 -5591.989} C_VEL
LIN {X 0,Y 511.102,Z 544.083,A -85,B 0,C 180,E1 -5592.71,E2 -5592.71} C_VEL
LIN {X 0,Y 511.338,Z 531.559,A -85,B 0,C 180,E1 -5593.31,E2 -5593.31} C_VEL
LIN {X 0,Y 511.556,Z 519.07,A -85,B 0,C 180,E1 -5593.734,E2 -5593.734} C_VEL
LIN {X 0,Y 511.695,Z 506.544,A -85,B 0,C 180,E1 -5594.009,E2 -5594.009} C_VEL
LIN {X 0,Y 512.131,Z 416.929,A -85,B 0,C 180,E1 -5595.334,E2 -5595.334} C_VEL
LIN {X 0,Y 509.882,Z 409.976,A -85,B 0,C 180,E1 -5595.531,E2 -5595.531} C_VEL
LIN {X 0,Y 509.841,Z 409.976,A -85,B 0,C 180,E1 -5598.485,E2 -5598.485} C_VEL
LIN {X 0,Y 509.849,Z 409.977,A -85,B 0,C 180,E1 -5601.002,E2 -5601.002} C_VEL
LIN {X 0,Y 509.822,Z 409.98,A -85,B 0,C 180,E1 -5603.564,E2 -5603.564} C_VEL
LIN {X 0,Y 509.881,Z 409.967,A -85,B 0,C 180,E1 -5606.371,E2 -5606.371} C_VEL
LIN {X 0,Y 509.875,Z 409.97,A -85,B 0,C 180,E1 -5608.845,E2 -5608.845} C_VEL
LIN {X 0,Y 509.823,Z 409.974,A -85,B 0,C 180,E1 -5611.59,E2 -5611.59} C_VEL
LIN {X 0,Y 509.85,Z 409.965,A -85,B 0,C 180,E1 -5614.414,E2 -5614.414} C_VEL
LIN {X 0,Y 509.82,Z 409.98,A -85,B 0,C 180,E1 -5617.341,E2 -5617.341} C_VEL
LIN {X 0,Y 509.825,Z 409.97,A -85,B 0,C 180,E1 -5620.075,E2 -5620.075} C_VEL
LIN {X 0,Y 509.177,Z 410.056,A -85,B 0,C 180,E1 -5620.735,E2 -5620.735} C_VEL
LIN {X 0,Y 506.326,Z 410.414,A -85,B 0,C 180,E1 -5621.806,E2 -5621.806} C_VEL
LIN {X 0,Y 503.9,Z 410.718,A -85,B 0,C 180,E1 -5622.668,E2 -5622.668} C_VEL
LIN {X 0,Y 502.854,Z 410.848,A -85,B 0,C 180,E1 -5623.334,E2 -5623.334} C_VEL
LIN {X 0,Y 502.767,Z 410.856,A -85,B 0,C 180,E1 -5623.56,E2 -5623.56} C_VEL
LIN {X 0,Y 502.793,Z 410.845,A -85,B 0,C 180,E1 -5625.661,E2 -5625.661} C_VEL
LIN {X 0,Y 502.821,Z 410.849,A -85,B 0,C 180,E1 -5629.005,E2 -5629.005} C_VEL
LIN {X 0,Y 502.793,Z 410.853,A -85,B 0,C 180,E1 -5632.046,E2 -5632.046} C_VEL
LIN {X 0,Y 502.8,Z 410.852,A -85,B 0,C 180,E1 -5635.034,E2 -5635.034} C_VEL
LIN {X 0,Y 502.786,Z 410.855,A -85,B 0,C 180,E1 -5637.915,E2 -5637.915} C_VEL
LIN {X 0,Y 502.807,Z 410.857,A -85,B 0,C 180,E1 -5640.711,E2 -5640.711} C_VEL
LIN {X 0,Y 502.776,Z 410.859,A -85,B 0,C 180,E1 -5643.46,E2 -5643.46} C_VEL
LIN {X 0,Y 502.82,Z 411.043,A -85,B 0,C 180,E1 -5644.988,E2 -5644.988} C_VEL
LIN {X 0,Y 504.611,Z 420.488,A -85,B 0,C 180,E1 -5646.547,E2 -5646.547} C_VEL
LIN {X 0,Y 504.288,Z 436.159,A -85,B 0,C 180,E1 -5649.027,E2 -5649.027} C_VEL
LIN {X 0,Y 503.839,Z 454.188,A -85,B 0,C 180,E1 -5651.83,E2 -5651.83} C_VEL
LIN {X 0,Y 503.525,Z 470.321,A -85,B 0,C 180,E1 -5654.245,E2 -5654.245} C_VEL
LIN {X 0,Y 505.406,Z 482.138,A -85,B 0,C 180,E1 -5654.48,E2 -5654.48} C_VEL
LIN {X 0,Y 504.877,Z 578.547,A -85,B 0,C 180,E1 -5655.875,E2 -5655.875} C_VEL
LIN {X 0,Y 504.632,Z 592.137,A -85,B 0,C 180,E1 -5656.228,E2 -5656.228} C_VEL
LIN {X 0,Y 504.383,Z 604.247,A -85,B 0,C 180,E1 -5656.708,E2 -5656.708} C_VEL
LIN {X 0,Y 504.066,Z 616.426,A -85,B 0,C 180,E1 -5657.362,E2 -5657.362} C_VEL
LIN {X 0,Y 503.784,Z 627.478,A -85,B 0,C 180,E1 -5658.125,E2 -5658.125} C_VEL
LIN {X 0,Y 503.354,Z 637.932,A -85,B 0,C 180,E1 -5659.033,E2 -5659.033} C_VEL
LIN {X 0,Y 502.97,Z 648.224,A -85,B 0,C 180,E1 -5660.144,E2 -5660.144} C_VEL
LIN {X 0,Y 502.707,Z 657.161,A -85,B 0,C 180,E1 -5661.356,E2 -5661.356} C_VEL
LIN {X 0,Y 502.437,Z 664.336,A -85,B 0,C 180,E1 -5662.566,E2 -5662.566} C_VEL
LIN {X 0,Y 502.357,Z 670.922,A -85,B 0,C 180,E1 -5663.977,E2 -5663.977} C_VEL
LIN {X 0,Y 502.116,Z 675.254,A -85,B 0,C 180,E1 -5665.183,E2 -5665.183} C_VEL
LIN {X 0,Y 502.236,Z 677.527,A -85,B 0,C 180,E1 -5665.988,E2 -5665.988} C_VEL
LIN {X 0,Y 502.124,Z 679.388,A -85,B 0,C 180,E1 -5666.791,E2 -5666.791} C_VEL
LIN {X 0,Y 502.121,Z 680.811,A -85,B 0,C 180,E1 -5667.593,E2 -5667.593} C_VEL
LIN {X 0,Y 501.991,Z 682.426,A -85,B 0,C 180,E1 -5669.198,E2 -5669.198} C_VEL
LIN {X 0,Y 501.98,Z 682.665,A -85,B 0,C 180,E1 -5670,E2 -5670} C_VEL
LIN {X 0,Y 501.99,Z 682.479,A -85,B 0,C 180,E1 -5670.802,E2 -5670.802} C_VEL
LIN {X 0,Y 502.121,Z 680.933,A -85,B 0,C 180,E1 -5672.407,E2 -5672.407} C_VEL
LIN {X 0,Y 502.125,Z 679.577,A -85,B 0,C 180,E1 -5673.209,E2 -5673.209} C_VEL
LIN {X 0,Y 502.189,Z 676.719,A -85,B 0,C 180,E1 -5674.414,E2 -5674.414} C_VEL
LIN {X 0,Y 502.289,Z 672.836,A -85,B 0,C 180,E1 -5675.621,E2 -5675.621} C_VEL
LIN {X 0,Y 502.356,Z 667.811,A -85,B 0,C 180,E1 -5676.829,E2 -5676.829} C_VEL
LIN {X 0,Y 502.561,Z 661.467,A -85,B 0,C 180,E1 -5678.039,E2 -5678.039} C_VEL
LIN {X 0,Y 502.773,Z 653.591,A -85,B 0,C 180,E1 -5679.251,E2 -5679.251} C_VEL
LIN {X 0,Y 503.059,Z 645.548,A -85,B 0,C 180,E1 -5680.261,E2 -5680.261} C_VEL
LIN {X 0,Y 503.46,Z 635.681,A -85,B 0,C 180,E1 -5681.27,E2 -5681.27} C_VEL
LIN {X 0,Y 503.827,Z 624.481,A -85,B 0,C 180,E1 -5682.189,E2 -5682.189} C_VEL
LIN {X 0,Y 504.152,Z 613.778,A -85,B 0,C 180,E1 -5682.888,E2 -5682.888} C_VEL
LIN {X 0,Y 504.437,Z 601.712,A -85,B 0,C 180,E1 -5683.495,E2 -5683.495} C_VEL
LIN {X 0,Y 504.745,Z 588.441,A -85,B 0,C 180,E1 -5683.975,E2 -5683.975} C_VEL
LIN {X 0,Y 504.913,Z 576.645,A -85,B 0,C 180,E1 -5684.253,E2 -5684.253} C_VEL
LIN {X 0,Y 505.392,Z 481.46,A -85,B 0,C 180,E1 -5685.62,E2 -5685.62} C_VEL
LIN {X 0,Y 503.554,Z 470.243,A -85,B 0,C 180,E1 -5685.849,E2 -5685.849} C_VEL
LIN {X 0,Y 503.926,Z 451.265,A -85,B 0,C 180,E1 -5688.71,E2 -5688.71} C_VEL
LIN {X 0,Y 504.455,Z 431.008,A -85,B 0,C 180,E1 -5691.881,E2 -5691.881} C_VEL
LIN {X 0,Y 504.533,Z 419.885,A -85,B 0,C 180,E1 -5693.64,E2 -5693.64} C_VEL
LIN {X 0,Y 502.784,Z 410.859,A -85,B 0,C 180,E1 -5695.174,E2 -5695.174} C_VEL
LIN {X 0,Y 502.776,Z 410.855,A -85,B 0,C 180,E1 -5698.377,E2 -5698.377} C_VEL
LIN {X 0,Y 502.795,Z 410.856,A -85,B 0,C 180,E1 -5701.144,E2 -5701.144} C_VEL
LIN {X 0,Y 502.806,Z 410.854,A -85,B 0,C 180,E1 -5703.994,E2 -5703.994} C_VEL
LIN {X 0,Y 502.768,Z 410.861,A -85,B 0,C 180,E1 -5707.176,E2 -5707.176} C_VEL
LIN {X 0,Y 502.791,Z 410.849,A -85,B 0,C 180,E1 -5710.015,E2 -5710.015} C_VEL
LIN {X 0,Y 502.806,Z 410.85,A -85,B 0,C 180,E1 -5712.199,E2 -5712.199} C_VEL
LIN {X 0,Y 502.804,Z 410.854,A -85,B 0,C 180,E1 -5715.468,E2 -5715.468} C_VEL
LIN {X 0,Y 502.823,Z 410.851,A -85,B 0,C 180,E1 -5718.934,E2 -5718.934} C_VEL
LIN {X 0,Y 502.794,Z 410.851,A -85,B 0,C 180,E1 -5722.046,E2 -5722.046} C_VEL
LIN {X 0,Y 502.8,Z 410.853,A -85,B 0,C 180,E1 -5725.034,E2 -5725.034} C_VEL
LIN {X 0,Y 502.786,Z 410.853,A -85,B 0,C 180,E1 -5727.915,E2 -5727.915} C_VEL
LIN {X 0,Y 502.807,Z 410.855,A -85,B 0,C 180,E1 -5730.711,E2 -5730.711} C_VEL
LIN {X 0,Y 502.777,Z 410.855,A -85,B 0,C 180,E1 -5733.46,E2 -5733.46} C_VEL
